LIN {X 0,Y 474.599,Z 728.17,A -85,B 0,C 180,E1 -7141.218,E2 -7141.218} C_VEL
LIN {X 0,Y 474.621,Z 728.178,A -85,B 0,C 180,E1 -7144.242,E2 -7144.242} C_VEL
LIN {X 0,Y 474.591,Z 728.17,A -85,B 0,C 180,E1 -7147.384,E2 -7147.384} C_VEL
LIN {X 0,Y 474.618,Z 728.176,A -85,B 0,C 180,E1 -7150.658,E2 -7150.658} C_VEL
LIN {X 0,Y 474.601,Z 728.174,A -85,B 0,C 180,E1 -7153.481,E2 -7153.481} C_VEL
LIN {X 0,Y 474.593,Z 728.164,A -85,B 0,C 180,E1 -7156.52,E2 -7156.52} C_VEL
LIN {X 0,Y 474.618,Z 728.164,A -85,B 0,C 180,E1 -7159.342,E2 -7159.342} C_VEL
LIN {X 0,Y 474.591,Z 728.181,A -85,B 0,C 180,E1 -7162.616,E2 -7162.616} C_VEL
LIN {X 0,Y 474.621,Z 728.167,A -85,B 0,C 180,E1 -7165.758,E2 -7165.758} C_VEL
LIN {X 0,Y 474.599,Z 728.178,A -85,B 0,C 180,E1 -7168.782,E2 -7168.782} C_VEL
LIN {X 0,Y 474.646,Z 728.168,A -85,B 0,C 180,E1 -7171.717,E2 -7171.717} C_VEL
LIN {X 0,Y 474.655,Z 728.161,A -85,B 0,C 180,E1 -7174.582,E2 -7174.582} C_VEL
LIN {X 0,Y 474.603,Z 728.179,A -85,B 0,C 180,E1 -7177.355,E2 -7177.355} C_VEL
LIN {X 0,Y 474.656,Z 728.166,A -85,B 0,C 180,E1 -7180.09,E2 -7180.09} C_VEL
LIN {X 0,Y 474.641,Z 728.164,A -85,B 0,C 180,E1 -7182.774,E2 -7182.774} C_VEL
LIN {X 0,Y 474.655,Z 728.173,A -85,B 0,C 180,E1 -7185.421,E2 -7185.421} C_VEL
LIN {X 0,Y 474.707,Z 728.161,A -85,B 0,C 180,E1 -7188.038,E2 -7188.038} C_VEL
LIN {X 0,Y 474.729,Z 728.152,A -85,B 0,C 180,E1 -7191.486,E2 -7191.486} C_VEL
LIN {X 0,Y 474.773,Z 728.149,A -85,B 0,C 180,E1 -7194.052,E2 -7194.052} C_VEL
LIN {X 0,Y 474.897,Z 728.146,A -85,B 0,C 180,E1 -7197.455,E2 -7197.455} C_VEL
LIN {X 0,Y 474.913,Z 728.132,A -85,B 0,C 180,E1 -7200,E2 -7200} C_VEL
LIN {X 0,Y 474.896,Z 728.125,A -85,B 0,C 180,E1 -7202.545,E2 -7202.545} C_VEL
LIN {X 0,Y 474.774,Z 728.157,A -85,B 0,C 180,E1 -7205.948,E2 -7205.948} C_VEL
LIN {X 0,Y 474.73,Z 728.158,A -85,B 0,C 180,E1 -7208.513,E2 -7208.513} C_VEL
LIN {X 0,Y 474.706,Z 728.156,A -85,B 0,C 180,E1 -7211.962,E2 -7211.962} C_VEL
LIN {X 0,Y 474.702,Z 728.163,A -85,B 0,C 180,E1 -7215.455,E2 -7215.455} C_VEL
LIN {X 0,Y 474.668,Z 728.164,A -85,B 0,C 180,E1 -7219.01,E2 -7219.01} C_VEL
LIN {X 0,Y 474.593,Z 728.171,A -85,B 0,C 180,E1 -7221.729,E2 -7221.729} C_VEL
LIN {X 0,Y 474.661,Z 728.169,A -85,B 0,C 180,E1 -7224.493,E2 -7224.493} C_VEL
LIN {X 0,Y 474.7,Z 728.161,A -85,B 0,C 180,E1 -7227.339,E2 -7227.339} C_VEL
LIN {X 0,Y 474.606,Z 728.172,A -85,B 0,C 180,E1 -7230.81,E2 -7230.81} C_VEL
LIN {X 0,Y 474.64,Z 728.175,A -85,B 0,C 180,E1 -7233.984,E2 -7233.984} C_VEL
LIN {X 0,Y 474.576,Z 728.167,A -85,B 0,C 180,E1 -7236.9,E2 -7236.9} C_VEL
LIN {X 0,Y 474.651,Z 728.143,A -85,B 0,C 180,E1 -7239.651,E2 -7239.651} C_VEL
LIN {X 0,Y 474.616,Z 728.173,A -85,B 0,C 180,E1 -7242.934,E2 -7242.934} C_VEL
LIN {X 0,Y 474.61,Z 728.175,A -85,B 0,C 180,E1 -7245.895,E2 -7245.895} C_VEL
LIN {X 0,Y 474.629,Z 728.168,A -85,B 0,C 180,E1 -7249.041,E2 -7249.041} C_VEL
LIN {X 0,Y 474.612,Z 728.174,A -85,B 0,C 180,E1 -7251.704,E2 -7251.704} C_VEL
LIN {X 0,Y 474.631,Z 728.174,A -85,B 0,C 180,E1 -7254.726,E2 -7254.726} C_VEL
LIN {X 0,Y 474.638,Z 728.168,A -85,B 0,C 180,E1 -7257.788,E2 -7257.788} C_VEL
LIN {X 0,Y 474.625,Z 728.176,A -85,B 0,C 180,E1 -7260.884,E2 -7260.884} C_VEL
LIN {X 0,Y 474.661,Z 728.165,A -85,B 0,C 180,E1 -7263.628,E2 -7263.628} C_VEL
LIN {X 0,Y 474.654,Z 728.288,A -85,B 0,C 180,E1 -7266.436,E2 -7266.436} C_VEL
LIN {X 0,Y 475.974,Z 735.804,A -85,B 0,C 180,E1 -7268.11,E2 -7268.11} C_VEL
LIN {X 0,Y 475.496,Z 750.231,A -85,B 0,C 180,E1 -7271.075,E2 -7271.075} C_VEL
LIN {X 0,Y 474.91,Z 765.942,A -85,B 0,C 180,E1 -7274.261,E2 -7274.261} C_VEL
LIN {X 0,Y 474.578,Z 778.638,A -85,B 0,C 180,E1 -7276.784,E2 -7276.784} C_VEL
LIN {X 0,Y 475.05,Z 782.47,A -85,B 0,C 180,E1 -7276.903,E2 -7276.903} C_VEL
LIN {X 0,Y 476.424,Z 793.246,A -85,B 0,C 180,E1 -7277.104,E2 -7277.104} C_VEL
LIN {X 0,Y 476.124,Z 856.175,A -85,B 0,C 180,E1 -7278.074,E2 -7278.074} C_VEL
LIN {X 0,Y 475.856,Z 866.65,A -85,B 0,C 180,E1 -7278.364,E2 -7278.364} C_VEL
LIN {X 0,Y 475.632,Z 877.37,A -85,B 0,C 180,E1 -7278.817,E2 -7278.817} C_VEL
LIN {X 0,Y 475.292,Z 888.005,A -85,B 0,C 180,E1 -7279.456,E2 -7279.456} C_VEL
LIN {X 0,Y 474.98,Z 896.334,A -85,B 0,C 180,E1 -7280.095,E2 -7280.095} C_VEL
LIN {X 0,Y 474.712,Z 904.218,A -85,B 0,C 180,E1 -7280.842,E2 -7280.842} C_VEL
LIN {X 0,Y 474.417,Z 911.588,A -85,B 0,C 180,E1 -7281.695,E2 -7281.695} C_VEL
LIN {X 0,Y 474.217,Z 919.07,A -85,B 0,C 180,E1 -7282.763,E2 -7282.763} C_VEL
LIN {X 0,Y 474.006,Z 925.901,A -85,B 0,C 180,E1 -7284.043,E2 -7284.043} C_VEL
LIN {X 0,Y 473.815,Z 931.085,A -85,B 0,C 180,E1 -7285.321,E2 -7285.321} C_VEL
LIN {X 0,Y 473.832,Z 934.897,A -85,B 0,C 180,E1 -7286.599,E2 -7286.599} C_VEL
LIN {X 0,Y 473.727,Z 936.647,A -85,B 0,C 180,E1 -7287.449,E2 -7287.449} C_VEL
LIN {X 0,Y 473.693,Z 937.902,A -85,B 0,C 180,E1 -7288.3,E2 -7288.3} C_VEL
LIN {X 0,Y 473.686,Z 938.684,A -85,B 0,C 180,E1 -7289.15,E2 -7289.15} C_VEL
LIN {X 0,Y 473.666,Z 938.979,A -85,B 0,C 180,E1 -7290,E2 -7290} C_VEL
LIN {X 0,Y 473.686,Z 938.683,A -85,B 0,C 180,E1 -7290.85,E2 -7290.85} C_VEL
LIN {X 0,Y 473.693,Z 937.901,A -85,B 0,C 180,E1 -7291.7,E2 -7291.7} C_VEL
LIN {X 0,Y 473.727,Z 936.646,A -85,B 0,C 180,E1 -7292.551,E2 -7292.551} C_VEL
LIN {X 0,Y 473.849,Z 933.739,A -85,B 0,C 180,E1 -7293.827,E2 -7293.827} C_VEL
LIN {X 0,Y 473.815,Z 931.085,A -85,B 0,C 180,E1 -7294.679,E2 -7294.679} C_VEL
LIN {X 0,Y 474.006,Z 925.898,A -85,B 0,C 180,E1 -7295.957,E2 -7295.957} C_VEL
LIN {X 0,Y 474.19,Z 919.063,A -85,B 0,C 180,E1 -7297.237,E2 -7297.237} C_VEL
LIN {X 0,Y 474.417,Z 911.591,A -85,B 0,C 180,E1 -7298.305,E2 -7298.305} C_VEL
LIN {X 0,Y 474.712,Z 904.224,A -85,B 0,C 180,E1 -7299.158,E2 -7299.158} C_VEL
LIN {X 0,Y 474.98,Z 896.337,A -85,B 0,C 180,E1 -7299.905,E2 -7299.905} C_VEL
LIN {X 0,Y 475.292,Z 888.006,A -85,B 0,C 180,E1 -7300.544,E2 -7300.544} C_VEL
LIN {X 0,Y 475.646,Z 877.374,A -85,B 0,C 180,E1 -7301.182,E2 -7301.182} C_VEL
LIN {X 0,Y 475.886,Z 865.822,A -85,B 0,C 180,E1 -7301.662,E2 -7301.662} C_VEL
LIN {X 0,Y 476.121,Z 856.176,A -85,B 0,C 180,E1 -7301.926,E2 -7301.926} C_VEL
LIN {X 0,Y 476.367,Z 808.389,A -85,B 0,C 180,E1 -7302.669,E2 -7302.669} C_VEL
LIN {X 0,Y 476.334,Z 792.236,A -85,B 0,C 180,E1 -7302.914,E2 -7302.914} C_VEL
LIN {X 0,Y 474.578,Z 778.937,A -85,B 0,C 180,E1 -7303.189,E2 -7303.189} C_VEL
LIN {X 0,Y 474.708,Z 773.874,A -85,B 0,C 180,E1 -7304.139,E2 -7304.139} C_VEL
LIN {X 0,Y 475.222,Z 757.609,A -85,B 0,C 180,E1 -7307.426,E2 -7307.426} C_VEL
LIN {X 0,Y 475.836,Z 741.257,A -85,B 0,C 180,E1 -7310.761,E2 -7310.761} C_VEL
LIN {X 0,Y 475.962,Z 735.791,A -85,B 0,C 180,E1 -7311.891,E2 -7311.891} C_VEL
LIN {X 0,Y 474.664,Z 728.224,A -85,B 0,C 180,E1 -7313.593,E2 -7313.593} C_VEL
LIN {X 0,Y 474.661,Z 728.165,A -85,B 0,C 180,E1 -7316.372,E2 -7316.372} C_VEL
LIN {X 0,Y 474.623,Z 728.174,A -85,B 0,C 180,E1 -7319.252,E2 -7319.252} C_VEL
LIN {X 0,Y 474.618,Z 728.171,A -85,B 0,C 180,E1 -7322.431,E2 -7322.431} C_VEL
LIN {X 0,Y 474.621,Z 728.174,A -85,B 0,C 180,E1 -7325.47,E2 -7325.47} C_VEL
LIN {X 0,Y 474.613,Z 728.173,A -85,B 0,C 180,E1 -7328.457,E2 -7328.457} C_VEL
LIN {X 0,Y 474.629,Z 728.167,A -85,B 0,C 180,E1 -7330.959,E2 -7330.959} C_VEL
LIN {X 0,Y 474.61,Z 728.175,A -85,B 0,C 180,E1 -7334.105,E2 -7334.105} C_VEL
LIN {X 0,Y 474.616,Z 728.172,A -85,B 0,C 180,E1 -7337.066,E2 -7337.066} C_VEL
LIN {X 0,Y 474.67,Z 728.139,A -85,B 0,C 180,E1 -7340.457,E2 -7340.457} C_VEL
LIN {X 0,Y 474.595,Z 728.172,A -85,B 0,C 180,E1 -7343.677,E2 -7343.677} C_VEL
LIN {X 0,Y 474.644,Z 728.169,A -85,B 0,C 180,E1 -7346.78,E2 -7346.78} C_VEL
LIN {X 0,Y 474.607,Z 728.175,A -85,B 0,C 180,E1 -7349.77,E2 -7349.77} C_VEL
LIN {X 0,Y 474.698,Z 728.162,A -85,B 0,C 180,E1 -7352.68,E2 -7352.68} C_VEL
LIN {X 0,Y 474.661,Z 728.169,A -85,B 0,C 180,E1 -7355.507,E2 -7355.507} C_VEL
LIN {X 0,Y 474.673,Z 728.156,A -85,B 0,C 180,E1 -7359.186,E2 -7359.186} C_VEL
LIN {X 0,Y 474.659,Z 728.17,A -85,B 0,C 180,E1 -7361.885,E2 -7361.885} C_VEL
LIN {X 0,Y 474.702,Z 728.163,A -85,B 0,C 180,E1 -7364.545,E2 -7364.545} C_VEL
LIN {X 0,Y 474.706,Z 728.155,A -85,B 0,C 180,E1 -7368.038,E2 -7368.038} C_VEL
LIN {X 0,Y 474.73,Z 728.157,A -85,B 0,C 180,E1 -7371.487,E2 -7371.487} C_VEL
LIN {X 0,Y 474.775,Z 728.156,A -85,B 0,C 180,E1 -7374.052,E2 -7374.052} C_VEL
LIN {X 0,Y 474.897,Z 728.124,A -85,B 0,C 180,E1 -7377.455,E2 -7377.455} C_VEL
LIN {X 0,Y 474.914,Z 728.132,A -85,B 0,C 180,E1 -7380,E2 -7380} C_VEL
LIN {X 0,Y 474.897,Z 728.145,A -85,B 0,C 180,E1 -7382.545,E2 -7382.545} C_VEL
LIN {X 0,Y 474.773,Z 728.148,A -85,B 0,C 180,E1 -7385.948,E2 -7385.948} C_VEL
LIN {X 0,Y 474.729,Z 728.151,A -85,B 0,C 180,E1 -7388.514,E2 -7388.514} C_VEL
LIN {X 0,Y 474.707,Z 728.161,A -85,B 0,C 180,E1 -7391.962,E2 -7391.962} C_VEL
LIN {X 0,Y 474.702,Z 728.157,A -85,B 0,C 180,E1 -7395.456,E2 -7395.456} C_VEL
LIN {X 0,Y 474.665,Z 728.169,A -85,B 0,C 180,E1 -7399.01,E2 -7399.01} C_VEL
LIN {X 0,Y 474.59,Z 728.176,A -85,B 0,C 180,E1 -7401.729,E2 -7401.729} C_VEL
LIN {X 0,Y 474.651,Z 728.167,A -85,B 0,C 180,E1 -7404.493,E2 -7404.493} C_VEL
LIN {X 0,Y 474.683,Z 728.167,A -85,B 0,C 180,E1 -7407.334,E2 -7407.334} C_VEL
LIN {X 0,Y 474.606,Z 728.174,A -85,B 0,C 180,E1 -7410.23,E2 -7410.23} C_VEL
LIN {X 0,Y 474.626,Z 728.171,A -85,B 0,C 180,E1 -7413.221,E2 -7413.221} C_VEL
LIN {X 0,Y 474.59,Z 728.176,A -85,B 0,C 180,E1 -7416.324,E2 -7416.324} C_VEL
LIN {X 0,Y 474.619,Z 728.168,A -85,B 0,C 180,E1 -7419.646,E2 -7419.646} C_VEL
LIN {X 0,Y 474.604,Z 728.149,A -85,B 0,C 180,E1 -7422.234,E2 -7422.234} C_VEL
LIN {X 0,Y 474.618,Z 728.17,A -85,B 0,C 180,E1 -7425.298,E2 -7425.298} C_VEL
LIN {X 0,Y 474.622,Z 728.173,A -85,B 0,C 180,E1 -7428.215,E2 -7428.215} C_VEL
LIN {X 0,Y 474.613,Z 728.168,A -85,B 0,C 180,E1 -7431.543,E2 -7431.543} C_VEL
LIN {X 0,Y 474.624,Z 728.173,A -85,B 0,C 180,E1 -7434.726,E2 -7434.726} C_VEL
LIN {X 0,Y 474.636,Z 728.169,A -85,B 0,C 180,E1 -7437.788,E2 -7437.788} C_VEL
LIN {X 0,Y 474.608,Z 728.175,A -85,B 0,C 180,E1 -7440.888,E2 -7440.888} C_VEL
LIN {X 0,Y 474.615,Z 728.18,A -85,B 0,C 180,E1 -7443.626,E2 -7443.626} C_VEL
LIN {X 0,Y 474.636,Z 728.17,A -85,B 0,C 180,E1 -7446.642,E2 -7446.642} C_VEL
LIN {X 0,Y 474.674,Z 728.172,A -85,B 0,C 180,E1 -7450.09,E2 -7450.09} C_VEL
LIN {X 0,Y 474.695,Z 728.188,A -85,B 0,C 180,E1 -7450.387,E2 -7450.387} C_VEL
LIN {X 0,Y 474.548,Z 728.717,A -85,B 0,C 180,E1 -7450.744,E2 -7450.744} C_VEL
LIN {X 0,Y 473.678,Z 730.812,A -85,B 0,C 180,E1 -7451.298,E2 -7451.298} C_VEL
LIN {X 0,Y 468.563,Z 738.885,A -85,B 0,C 180,E1 -7453.14,E2 -7453.14} C_VEL
LIN {X 0,Y 467.847,Z 741.421,A -85,B 0,C 180,E1 -7453.786,E2 -7453.786} C_VEL
LIN {X 0,Y 467.504,Z 752.277,A -85,B 0,C 180,E1 -7456.526,E2 -7456.526} C_VEL
LIN {X 0,Y 467.554,Z 753.524,A -85,B 0,C 180,E1 -7456.689,E2 -7456.689} C_VEL
LIN {X 0,Y 469.574,Z 765.597,A -85,B 0,C 180,E1 -7456.949,E2 -7456.949} C_VEL
LIN {X 0,Y 469.229,Z 828.139,A -85,B 0,C 180,E1 -7457.923,E2 -7457.923} C_VEL
LIN {X 0,Y 469.116,Z 837.235,A -85,B 0,C 180,E1 -7458.167,E2 -7458.167} C_VEL
LIN {X 0,Y 468.858,Z 846.827,A -85,B 0,C 180,E1 -7458.544,E2 -7458.544} C_VEL
LIN {X 0,Y 468.61,Z 856.862,A -85,B 0,C 180,E1 -7459.085,E2 -7459.085} C_VEL
LIN {X 0,Y 468.208,Z 867.274,A -85,B 0,C 180,E1 -7459.841,E2 -7459.841} C_VEL
LIN {X 0,Y 467.908,Z 875.411,A -85,B 0,C 180,E1 -7460.599,E2 -7460.599} C_VEL
LIN {X 0,Y 467.607,Z 882.124,A -85,B 0,C 180,E1 -7461.356,E2 -7461.356} C_VEL
LIN {X 0,Y 467.352,Z 888.477,A -85,B 0,C 180,E1 -7462.222,E2 -7462.222} C_VEL
LIN {X 0,Y 467.173,Z 894.148,A -85,B 0,C 180,E1 -7463.161,E2 -7463.161} C_VEL
LIN {X 0,Y 467.132,Z 898.161,A -85,B 0,C 180,E1 -7463.955,E2 -7463.955} C_VEL
LIN {X 0,Y 466.829,Z 901.837,A -85,B 0,C 180,E1 -7464.817,E2 -7464.817} C_VEL
LIN {X 0,Y 466.84,Z 904.829,A -85,B 0,C 180,E1 -7465.683,E2 -7465.683} C_VEL
LIN {X 0,Y 466.793,Z 907.149,A -85,B 0,C 180,E1 -7466.547,E2 -7466.547} C_VEL
LIN {X 0,Y 466.687,Z 908.919,A -85,B 0,C 180,E1 -7467.411,E2 -7467.411} C_VEL
LIN {X 0,Y 466.634,Z 910.196,A -85,B 0,C 180,E1 -7468.274,E2 -7468.274} C_VEL
LIN {X 0,Y 466.617,Z 911.003,A -85,B 0,C 180,E1 -7469.137,E2 -7469.137} C_VEL
LIN {X 0,Y 466.597,Z 911.311,A -85,B 0,C 180,E1 -7470,E2 -7470} C_VEL
LIN {X 0,Y 466.617,Z 911.037,A -85,B 0,C 180,E1 -7470.863,E2 -7470.863} C_VEL
LIN {X 0,Y 466.634,Z 910.296,A -85,B 0,C 180,E1 -7471.726,E2 -7471.726} C_VEL
LIN {X 0,Y 466.687,Z 909.088,A -85,B 0,C 180,E1 -7472.589,E2 -7472.589} C_VEL
LIN {X 0,Y 466.841,Z 906.243,A -85,B 0,C 180,E1 -7473.884,E2 -7473.884} C_VEL
LIN {X 0,Y 466.806,Z 903.66,A -85,B 0,C 180,E1 -7474.75,E2 -7474.75} C_VEL
LIN {X 0,Y 467.107,Z 898.559,A -85,B 0,C 180,E1 -7476.046,E2 -7476.046} C_VEL
LIN {X 0,Y 467.194,Z 893.079,A -85,B 0,C 180,E1 -7477.129,E2 -7477.129} C_VEL
LIN {X 0,Y 467.46,Z 886.192,A -85,B 0,C 180,E1 -7478.211,E2 -7478.211} C_VEL
LIN {X 0,Y 467.806,Z 878.281,A -85,B 0,C 180,E1 -7479.185,E2 -7479.185} C_VEL
LIN {X 0,Y 468.108,Z 870.734,A -85,B 0,C 180,E1 -7479.942,E2 -7479.942} C_VEL
LIN {X 0,Y 468.366,Z 862.827,A -85,B 0,C 180,E1 -7480.592,E2 -7480.592} C_VEL
LIN {X 0,Y 468.66,Z 854.66,A -85,B 0,C 180,E1 -7481.132,E2 -7481.132} C_VEL
LIN {X 0,Y 468.943,Z 846.391,A -85,B 0,C 180,E1 -7481.563,E2 -7481.563} C_VEL
LIN {X 0,Y 469.105,Z 837.469,A -85,B 0,C 180,E1 -7481.915,E2 -7481.915} C_VEL
LIN {X 0,Y 469.271,Z 828.375,A -85,B 0,C 180,E1 -7482.161,E2 -7482.161} C_VEL
LIN {X 0,Y 469.463,Z 764.852,A -85,B 0,C 180,E1 -7483.156,E2 -7483.156} C_VEL
LIN {X 0,Y 467.486,Z 752.928,A -85,B 0,C 180,E1 -7483.398,E2 -7483.398} C_VEL
LIN {X 0,Y 467.842,Z 741.837,A -85,B 0,C 180,E1 -7486.197,E2 -7486.197} C_VEL
LIN {X 0,Y 468.105,Z 733.408,A -85,B 0,C 180,E1 -7488.378,E2 -7488.378} C_VEL
LIN {X 0,Y 467.664,Z 729.117,A -85,B 0,C 180,E1 -7489.591,E2 -7489.591} C_VEL
LIN {X 0,Y 467.577,Z 729.049,A -85,B 0,C 180,E1 -7493.004,E2 -7493.004} C_VEL
LIN {X 0,Y 467.569,Z 729.056,A -85,B 0,C 180,E1 -7495.842,E2 -7495.842} C_VEL
LIN {X 0,Y 467.555,Z 729.056,A -85,B 0,C 180,E1 -7498.751,E2 -7498.751} C_VEL
LIN {X 0,Y 467.583,Z 729.045,A -85,B 0,C 180,E1 -7501.74,E2 -7501.74} C_VEL
LIN {X 0,Y 467.56,Z 729.057,A -85,B 0,C 180,E1 -7504.833,E2 -7504.833} C_VEL
LIN {X 0,Y 467.565,Z 729.047,A -85,B 0,C 180,E1 -7508.045,E2 -7508.045} C_VEL
LIN {X 0,Y 467.579,Z 729.05,A -85,B 0,C 180,E1 -7511.277,E2 -7511.277} C_VEL
LIN {X 0,Y 467.553,Z 729.052,A -85,B 0,C 180,E1 -7513.821,E2 -7513.821} C_VEL
LIN {X 0,Y 467.55,Z 729.046,A -85,B 0,C 180,E1 -7516.255,E2 -7516.255} C_VEL
LIN {X 0,Y 467.576,Z 729.04,A -85,B 0,C 180,E1 -7519.735,E2 -7519.735} C_VEL
LIN {X 0,Y 467.549,Z 729.061,A -85,B 0,C 180,E1 -7522.814,E2 -7522.814} C_VEL
LIN {X 0,Y 467.578,Z 729.045,A -85,B 0,C 180,E1 -7525.76,E2 -7525.76} C_VEL
LIN {X 0,Y 467.569,Z 729.057,A -85,B 0,C 180,E1 -7528.955,E2 -7528.955} C_VEL
LIN {X 0,Y 467.635,Z 729.042,A -85,B 0,C 180,E1 -7532.462,E2 -7532.462} C_VEL
LIN {X 0,Y 467.596,Z 729.046,A -85,B 0,C 180,E1 -7535.112,E2 -7535.112} C_VEL
LIN {X 0,Y 467.536,Z 729.055,A -85,B 0,C 180,E1 -7537.926,E2 -7537.926} C_VEL
LIN {X 0,Y 467.624,Z 729.044,A -85,B 0,C 180,E1 -7540.692,E2 -7540.692} C_VEL
LIN {X 0,Y 467.651,Z 729.034,A -85,B 0,C 180,E1 -7544.115,E2 -7544.115} C_VEL
LIN {X 0,Y 467.656,Z 729.043,A -85,B 0,C 180,E1 -7547.642,E2 -7547.642} C_VEL
LIN {X 0,Y 467.663,Z 729.034,A -85,B 0,C 180,E1 -7550.485,E2 -7550.485} C_VEL
LIN {X 0,Y 467.702,Z 729.024,A -85,B 0,C 180,E1 -7553.095,E2 -7553.095} C_VEL
LIN {X 0,Y 467.726,Z 729.027,A -85,B 0,C 180,E1 -7554.827,E2 -7554.827} C_VEL
LIN {X 0,Y 467.862,Z 729.021,A -85,B 0,C 180,E1 -7557.417,E2 -7557.417} C_VEL
LIN {X 0,Y 467.884,Z 729.008,A -85,B 0,C 180,E1 -7560,E2 -7560} C_VEL
LIN {X 0,Y 467.861,Z 729,A -85,B 0,C 180,E1 -7562.583,E2 -7562.583} C_VEL
LIN {X 0,Y 467.739,Z 729.032,A -85,B 0,C 180,E1 -7566.037,E2 -7566.037} C_VEL
LIN {X 0,Y 467.684,Z 729.035,A -85,B 0,C 180,E1 -7568.643,E2 -7568.643} C_VEL
LIN {X 0,Y 467.658,Z 729.032,A -85,B 0,C 180,E1 -7572.145,E2 -7572.145} C_VEL
LIN {X 0,Y 467.641,Z 729.045,A -85,B 0,C 180,E1 -7575.695,E2 -7575.695} C_VEL
LIN {X 0,Y 467.62,Z 729.042,A -85,B 0,C 180,E1 -7578.765,E2 -7578.765} C_VEL
LIN {X 0,Y 467.583,Z 729.04,A -85,B 0,C 180,E1 -7581.268,E2 -7581.268} C_VEL
LIN {X 0,Y 467.576,Z 729.053,A -85,B 0,C 180,E1 -7583.943,E2 -7583.943} C_VEL
LIN {X 0,Y 467.618,Z 729.044,A -85,B 0,C 180,E1 -7586.8,E2 -7586.8} C_VEL
LIN {X 0,Y 467.555,Z 729.047,A -85,B 0,C 180,E1 -7589.738,E2 -7589.738} C_VEL
LIN {X 0,Y 467.585,Z 729.05,A -85,B 0,C 180,E1 -7592.758,E2 -7592.758} C_VEL
LIN {X 0,Y 467.558,Z 729.053,A -85,B 0,C 180,E1 -7595.889,E2 -7595.889} C_VEL
LIN {X 0,Y 467.601,Z 729.019,A -85,B 0,C 180,E1 -7599.143,E2 -7599.143} C_VEL
LIN {X 0,Y 467.587,Z 729.05,A -85,B 0,C 180,E1 -7602.567,E2 -7602.567} C_VEL
LIN {X 0,Y 467.571,Z 729.051,A -85,B 0,C 180,E1 -7605.053,E2 -7605.053} C_VEL
LIN {X 0,Y 467.589,Z 729.042,A -85,B 0,C 180,E1 -7607.44,E2 -7607.44} C_VEL
LIN {X 0,Y 467.593,Z 729.052,A -85,B 0,C 180,E1 -7610.856,E2 -7610.856} C_VEL
LIN {X 0,Y 467.564,Z 729.051,A -85,B 0,C 180,E1 -7614.26,E2 -7614.26} C_VEL
LIN {X 0,Y 467.583,Z 729.047,A -85,B 0,C 180,E1 -7617.321,E2 -7617.321} C_VEL
LIN {X 0,Y 467.571,Z 729.05,A -85,B 0,C 180,E1 -7620.667,E2 -7620.667} C_VEL
LIN {X 0,Y 467.616,Z 729.042,A -85,B 0,C 180,E1 -7623.2,E2 -7623.2} C_VEL
LIN {X 0,Y 467.633,Z 729.209,A -85,B 0,C 180,E1 -7626.305,E2 -7626.305} C_VEL
LIN {X 0,Y 468.955,Z 736.728,A -85,B 0,C 180,E1 -7627.996,E2 -7627.996} C_VEL
LIN {X 0,Y 468.526,Z 749.812,A -85,B 0,C 180,E1 -7630.731,E2 -7630.731} C_VEL
LIN {X 0,Y 467.915,Z 765.671,A -85,B 0,C 180,E1 -7634.001,E2 -7634.001} C_VEL
LIN {X 0,Y 467.541,Z 778.521,A -85,B 0,C 180,E1 -7636.591,E2 -7636.591} C_VEL
LIN {X 0,Y 468.158,Z 783.277,A -85,B 0,C 180,E1 -7636.722,E2 -7636.722} C_VEL
LIN {X 0,Y 469.509,Z 795.019,A -85,B 0,C 180,E1 -7636.941,E2 -7636.941} C_VEL
LIN {X 0,Y 469.185,Z 855.966,A -85,B 0,C 180,E1 -7637.895,E2 -7637.895} C_VEL
LIN {X 0,Y 468.922,Z 866.441,A -85,B 0,C 180,E1 -7638.19,E2 -7638.19} C_VEL
LIN {X 0,Y 468.651,Z 877.161,A -85,B 0,C 180,E1 -7638.649,E2 -7638.649} C_VEL
LIN {X 0,Y 468.295,Z 887.796,A -85,B 0,C 180,E1 -7639.297,E2 -7639.297} C_VEL
LIN {X 0,Y 467.965,Z 896.124,A -85,B 0,C 180,E1 -7639.945,E2 -7639.945} C_VEL
LIN {X 0,Y 467.673,Z 904.008,A -85,B 0,C 180,E1 -7640.703,E2 -7640.703} C_VEL
LIN {X 0,Y 467.368,Z 911.379,A -85,B 0,C 180,E1 -7641.569,E2 -7641.569} C_VEL
LIN {X 0,Y 467.143,Z 918.86,A -85,B 0,C 180,E1 -7642.653,E2 -7642.653} C_VEL
LIN {X 0,Y 466.916,Z 925.691,A -85,B 0,C 180,E1 -7643.952,E2 -7643.952} C_VEL
LIN {X 0,Y 466.739,Z 930.876,A -85,B 0,C 180,E1 -7645.249,E2 -7645.249} C_VEL
LIN {X 0,Y 466.734,Z 934.687,A -85,B 0,C 180,E1 -7646.547,E2 -7646.547} C_VEL
LIN {X 0,Y 466.65,Z 936.438,A -85,B 0,C 180,E1 -7647.41,E2 -7647.41} C_VEL
LIN {X 0,Y 466.603,Z 937.693,A -85,B 0,C 180,E1 -7648.274,E2 -7648.274} C_VEL
LIN {X 0,Y 466.616,Z 938.476,A -85,B 0,C 180,E1 -7649.137,E2 -7649.137} C_VEL
LIN {X 0,Y 466.596,Z 938.771,A -85,B 0,C 180,E1 -7650,E2 -7650} C_VEL
LIN {X 0,Y 466.616,Z 938.475,A -85,B 0,C 180,E1 -7650.863,E2 -7650.863} C_VEL
LIN {X 0,Y 466.603,Z 937.692,A -85,B 0,C 180,E1 -7651.726,E2 -7651.726} C_VEL
LIN {X 0,Y 466.65,Z 936.437,A -85,B 0,C 180,E1 -7652.59,E2 -7652.59} C_VEL
LIN {X 0,Y 466.74,Z 933.529,A -85,B 0,C 180,E1 -7653.885,E2 -7653.885} C_VEL
LIN {X 0,Y 466.739,Z 930.876,A -85,B 0,C 180,E1 -7654.751,E2 -7654.751} C_VEL
LIN {X 0,Y 466.917,Z 925.688,A -85,B 0,C 180,E1 -7656.048,E2 -7656.048} C_VEL
LIN {X 0,Y 467.132,Z 918.853,A -85,B 0,C 180,E1 -7657.347,E2 -7657.347} C_VEL
LIN {X 0,Y 467.368,Z 911.381,A -85,B 0,C 180,E1 -7658.431,E2 -7658.431} C_VEL
LIN {X 0,Y 467.673,Z 904.015,A -85,B 0,C 180,E1 -7659.297,E2 -7659.297} C_VEL
LIN {X 0,Y 467.965,Z 896.127,A -85,B 0,C 180,E1 -7660.055,E2 -7660.055} C_VEL
LIN {X 0,Y 468.297,Z 887.797,A -85,B 0,C 180,E1 -7660.703,E2 -7660.703} C_VEL
LIN {X 0,Y 468.697,Z 877.166,A -85,B 0,C 180,E1 -7661.35,E2 -7661.35} C_VEL
LIN {X 0,Y 468.932,Z 865.613,A -85,B 0,C 180,E1 -7661.838,E2 -7661.838} C_VEL
LIN {X 0,Y 469.195,Z 855.968,A -85,B 0,C 180,E1 -7662.105,E2 -7662.105} C_VEL
LIN {X 0,Y 469.455,Z 793.148,A -85,B 0,C 180,E1 -7663.089,E2 -7663.089} C_VEL
LIN {X 0,Y 467.567,Z 778.882,A -85,B 0,C 180,E1 -7663.381,E2 -7663.381} C_VEL
LIN {X 0,Y 467.58,Z 776.934,A -85,B 0,C 180,E1 -7663.694,E2 -7663.694} C_VEL
LIN {X 0,Y 468.085,Z 761.783,A -85,B 0,C 180,E1 -7666.8,E2 -7666.8} C_VEL
LIN {X 0,Y 468.663,Z 746.541,A -85,B 0,C 180,E1 -7669.947,E2 -7669.947} C_VEL
LIN {X 0,Y 468.933,Z 736.714,A -85,B 0,C 180,E1 -7672.005,E2 -7672.005} C_VEL
LIN {X 0,Y 467.633,Z 729.106,A -85,B 0,C 180,E1 -7673.741,E2 -7673.741} C_VEL
LIN {X 0,Y 467.616,Z 729.042,A -85,B 0,C 180,E1 -7676.8,E2 -7676.8} C_VEL
LIN {X 0,Y 467.555,Z 729.047,A -85,B 0,C 180,E1 -7679.738,E2 -7679.738} C_VEL
LIN {X 0,Y 467.584,Z 729.049,A -85,B 0,C 180,E1 -7682.758,E2 -7682.758} C_VEL
LIN {X 0,Y 467.558,Z 729.051,A -85,B 0,C 180,E1 -7685.889,E2 -7685.889} C_VEL
LIN {X 0,Y 467.593,Z 729.052,A -85,B 0,C 180,E1 -7689.144,E2 -7689.144} C_VEL
LIN {X 0,Y 467.587,Z 729.043,A -85,B 0,C 180,E1 -7692.567,E2 -7692.567} C_VEL
LIN {X 0,Y 467.571,Z 729.052,A -85,B 0,C 180,E1 -7695.053,E2 -7695.053} C_VEL
LIN {X 0,Y 467.589,Z 729.05,A -85,B 0,C 180,E1 -7697.44,E2 -7697.44} C_VEL
LIN {X 0,Y 467.601,Z 729.018,A -85,B 0,C 180,E1 -7700.857,E2 -7700.857} C_VEL
LIN {X 0,Y 467.564,Z 729.051,A -85,B 0,C 180,E1 -7704.26,E2 -7704.26} C_VEL
LIN {X 0,Y 467.583,Z 729.051,A -85,B 0,C 180,E1 -7707.321,E2 -7707.321} C_VEL
LIN {X 0,Y 467.571,Z 729.043,A -85,B 0,C 180,E1 -7710.668,E2 -7710.668} C_VEL
LIN {X 0,Y 467.618,Z 729.044,A -85,B 0,C 180,E1 -7713.2,E2 -7713.2} C_VEL
LIN {X 0,Y 467.595,Z 729.045,A -85,B 0,C 180,E1 -7716.468,E2 -7716.468} C_VEL
LIN {X 0,Y 467.626,Z 729.038,A -85,B 0,C 180,E1 -7719.777,E2 -7719.777} C_VEL
LIN {X 0,Y 467.612,Z 729.049,A -85,B 0,C 180,E1 -7722.507,E2 -7722.507} C_VEL
LIN {X 0,Y 467.608,Z 729.042,A -85,B 0,C 180,E1 -7725.197,E2 -7725.197} C_VEL
LIN {X 0,Y 467.658,Z 729.031,A -85,B 0,C 180,E1 -7727.855,E2 -7727.855} C_VEL
LIN {X 0,Y 467.684,Z 729.035,A -85,B 0,C 180,E1 -7731.357,E2 -7731.357} C_VEL
LIN {X 0,Y 467.739,Z 729.032,A -85,B 0,C 180,E1 -7733.963,E2 -7733.963} C_VEL
LIN {X 0,Y 467.862,Z 729,A -85,B 0,C 180,E1 -7737.417,E2 -7737.417} C_VEL
LIN {X 0,Y 467.885,Z 729.007,A -85,B 0,C 180,E1 -7740,E2 -7740} C_VEL
LIN {X 0,Y 467.863,Z 729.022,A -85,B 0,C 180,E1 -7742.583,E2 -7742.583} C_VEL
LIN {X 0,Y 467.737,Z 729.025,A -85,B 0,C 180,E1 -7746.038,E2 -7746.038} C_VEL
LIN {X 0,Y 467.682,Z 729.031,A -85,B 0,C 180,E1 -7748.643,E2 -7748.643} C_VEL
LIN {X 0,Y 467.658,Z 729.04,A -85,B 0,C 180,E1 -7752.145,E2 -7752.145} C_VEL
LIN {X 0,Y 467.641,Z 729.035,A -85,B 0,C 180,E1 -7755.695,E2 -7755.695} C_VEL
LIN {X 0,Y 467.615,Z 729.042,A -85,B 0,C 180,E1 -7758.763,E2 -7758.763} C_VEL
LIN {X 0,Y 467.582,Z 729.053,A -85,B 0,C 180,E1 -7761.268,E2 -7761.268} C_VEL
LIN {X 0,Y 467.569,Z 729.047,A -85,B 0,C 180,E1 -7763.944,E2 -7763.944} C_VEL
LIN {X 0,Y 467.615,Z 729.04,A -85,B 0,C 180,E1 -7766.8,E2 -7766.8} C_VEL
LIN {X 0,Y 467.555,Z 729.053,A -85,B 0,C 180,E1 -7769.738,E2 -7769.738} C_VEL
LIN {X 0,Y 467.58,Z 729.048,A -85,B 0,C 180,E1 -7772.759,E2 -7772.759} C_VEL
LIN {X 0,Y 467.554,Z 729.053,A -85,B 0,C 180,E1 -7775.89,E2 -7775.89} C_VEL
LIN {X 0,Y 467.577,Z 729.053,A -85,B 0,C 180,E1 -7779.145,E2 -7779.145} C_VEL
LIN {X 0,Y 467.577,Z 729.033,A -85,B 0,C 180,E1 -7781.403,E2 -7781.403} C_VEL
LIN {X 0,Y 467.567,Z 729.045,A -85,B 0,C 180,E1 -7785.053,E2 -7785.053} C_VEL
LIN {X 0,Y 467.59,Z 729.055,A -85,B 0,C 180,E1 -7787.44,E2 -7787.44} C_VEL
LIN {X 0,Y 467.561,Z 729.045,A -85,B 0,C 180,E1 -7790.853,E2 -7790.853} C_VEL
LIN {X 0,Y 467.56,Z 729.055,A -85,B 0,C 180,E1 -7794.261,E2 -7794.261} C_VEL
LIN {X 0,Y 467.581,Z 729.053,A -85,B 0,C 180,E1 -7797.321,E2 -7797.321} C_VEL
LIN {X 0,Y 467.558,Z 729.053,A -85,B 0,C 180,E1 -7800.67,E2 -7800.67} C_VEL
LIN {X 0,Y 467.565,Z 729.053,A -85,B 0,C 180,E1 -7803.196,E2 -7803.196} C_VEL
LIN {X 0,Y 467.591,Z 729.048,A -85,B 0,C 180,E1 -7806.469,E2 -7806.469} C_VEL
LIN {X 0,Y 467.635,Z 729.05,A -85,B 0,C 180,E1 -7809.778,E2 -7809.778} C_VEL
LIN {X 0,Y 467.716,Z 729.213,A -85,B 0,C 180,E1 -7810.582,E2 -7810.582} C_VEL
LIN {X 0,Y 468.082,Z 734.779,A -85,B 0,C 180,E1 -7812.073,E2 -7812.073} C_VEL
LIN {X 0,Y 467.847,Z 741.421,A -85,B 0,C 180,E1 -7813.786,E2 -7813.786} C_VEL
LIN {X 0,Y 467.125,Z 743.198,A -85,B 0,C 180,E1 -7814.214,E2 -7814.214} C_VEL
LIN {X 0,Y 464.196,Z 746.192,A -85,B 0,C 180,E1 -7814.864,E2 -7814.864} C_VEL
LIN {X 0,Y 461.251,Z 749.201,A -85,B 0,C 180,E1 -7815.52,E2 -7815.52} C_VEL
LIN {X 0,Y 460.519,Z 751.004,A -85,B 0,C 180,E1 -7815.953,E2 -7815.953} C_VEL
LIN {X 0,Y 460.516,Z 753.153,A -85,B 0,C 180,E1 -7816.441,E2 -7816.441} C_VEL
LIN {X 0,Y 461.216,Z 757.471,A -85,B 0,C 180,E1 -7816.576,E2 -7816.576} C_VEL
LIN {X 0,Y 462.71,Z 766.919,A -85,B 0,C 180,E1 -7816.769,E2 -7816.769} C_VEL
LIN {X 0,Y 462.301,Z 828.374,A -85,B 0,C 180,E1 -7817.74,E2 -7817.74} C_VEL
LIN {X 0,Y 462.198,Z 837.461,A -85,B 0,C 180,E1 -7817.987,E2 -7817.987} C_VEL
LIN {X 0,Y 461.905,Z 847.048,A -85,B 0,C 180,E1 -7818.369,E2 -7818.369} C_VEL
LIN {X 0,Y 461.648,Z 857.08,A -85,B 0,C 180,E1 -7818.919,E2 -7818.919} C_VEL
LIN {X 0,Y 461.235,Z 867.489,A -85,B 0,C 180,E1 -7819.686,E2 -7819.686} C_VEL
LIN {X 0,Y 460.922,Z 875.625,A -85,B 0,C 180,E1 -7820.455,E2 -7820.455} C_VEL
LIN {X 0,Y 460.582,Z 882.338,A -85,B 0,C 180,E1 -7821.223,E2 -7821.223} C_VEL
LIN {X 0,Y 460.335,Z 888.69,A -85,B 0,C 180,E1 -7822.102,E2 -7822.102} C_VEL
LIN {X 0,Y 460.112,Z 894.822,A -85,B 0,C 180,E1 -7823.142,E2 -7823.142} C_VEL
LIN {X 0,Y 460.073,Z 898.372,A -85,B 0,C 180,E1 -7823.862,E2 -7823.862} C_VEL
LIN {X 0,Y 459.777,Z 902.048,A -85,B 0,C 180,E1 -7824.738,E2 -7824.738} C_VEL
LIN {X 0,Y 459.748,Z 905.041,A -85,B 0,C 180,E1 -7825.616,E2 -7825.616} C_VEL
LIN {X 0,Y 459.732,Z 907.359,A -85,B 0,C 180,E1 -7826.494,E2 -7826.494} C_VEL
LIN {X 0,Y 459.611,Z 909.129,A -85,B 0,C 180,E1 -7827.371,E2 -7827.371} C_VEL
LIN {X 0,Y 459.545,Z 910.405,A -85,B 0,C 180,E1 -7828.247,E2 -7828.247} C_VEL
LIN {X 0,Y 459.521,Z 911.212,A -85,B 0,C 180,E1 -7829.124,E2 -7829.124} C_VEL
LIN {X 0,Y 459.528,Z 911.519,A -85,B 0,C 180,E1 -7830,E2 -7830} C_VEL
LIN {X 0,Y 459.521,Z 911.245,A -85,B 0,C 180,E1 -7830.876,E2 -7830.876} C_VEL
LIN {X 0,Y 459.546,Z 910.504,A -85,B 0,C 180,E1 -7831.753,E2 -7831.753} C_VEL
LIN {X 0,Y 459.611,Z 909.295,A -85,B 0,C 180,E1 -7832.629,E2 -7832.629} C_VEL
LIN {X 0,Y 459.774,Z 906.45,A -85,B 0,C 180,E1 -7833.944,E2 -7833.944} C_VEL
LIN {X 0,Y 459.724,Z 903.867,A -85,B 0,C 180,E1 -7834.823,E2 -7834.823} C_VEL
LIN {X 0,Y 460.062,Z 898.765,A -85,B 0,C 180,E1 -7836.139,E2 -7836.139} C_VEL
LIN {X 0,Y 460.149,Z 893.284,A -85,B 0,C 180,E1 -7837.239,E2 -7837.239} C_VEL
LIN {X 0,Y 460.441,Z 886.397,A -85,B 0,C 180,E1 -7838.338,E2 -7838.338} C_VEL
LIN {X 0,Y 460.81,Z 878.483,A -85,B 0,C 180,E1 -7839.326,E2 -7839.326} C_VEL
LIN {X 0,Y 461.104,Z 870.937,A -85,B 0,C 180,E1 -7840.095,E2 -7840.095} C_VEL
LIN {X 0,Y 461.39,Z 863.028,A -85,B 0,C 180,E1 -7840.754,E2 -7840.754} C_VEL
LIN {X 0,Y 461.703,Z 854.859,A -85,B 0,C 180,E1 -7841.302,E2 -7841.302} C_VEL
LIN {X 0,Y 461.993,Z 846.587,A -85,B 0,C 180,E1 -7841.74,E2 -7841.74} C_VEL
LIN {X 0,Y 462.181,Z 837.66,A -85,B 0,C 180,E1 -7842.097,E2 -7842.097} C_VEL
LIN {X 0,Y 462.346,Z 828.659,A -85,B 0,C 180,E1 -7842.343,E2 -7842.343} C_VEL
LIN {X 0,Y 462.613,Z 765.973,A -85,B 0,C 180,E1 -7843.339,E2 -7843.339} C_VEL
LIN {X 0,Y 460.479,Z 752.975,A -85,B 0,C 180,E1 -7843.632,E2 -7843.632} C_VEL
LIN {X 0,Y 460.856,Z 742.21,A -85,B 0,C 180,E1 -7846.393,E2 -7846.393} C_VEL
LIN {X 0,Y 461.049,Z 733.57,A -85,B 0,C 180,E1 -7848.67,E2 -7848.67} C_VEL
LIN {X 0,Y 460.627,Z 730.016,A -85,B 0,C 180,E1 -7849.671,E2 -7849.671} C_VEL
LIN {X 0,Y 460.545,Z 729.925,A -85,B 0,C 180,E1 -7853.376,E2 -7853.376} C_VEL
LIN {X 0,Y 460.521,Z 729.935,A -85,B 0,C 180,E1 -7856.268,E2 -7856.268} C_VEL
LIN {X 0,Y 460.527,Z 729.929,A -85,B 0,C 180,E1 -7859.232,E2 -7859.232} C_VEL
LIN {X 0,Y 460.531,Z 729.925,A -85,B 0,C 180,E1 -7862.284,E2 -7862.284} C_VEL
LIN {X 0,Y 460.509,Z 729.932,A -85,B 0,C 180,E1 -7865.446,E2 -7865.446} C_VEL
LIN {X 0,Y 460.534,Z 729.921,A -85,B 0,C 180,E1 -7868.896,E2 -7868.896} C_VEL
LIN {X 0,Y 460.524,Z 729.931,A -85,B 0,C 180,E1 -7872.181,E2 -7872.181} C_VEL
LIN {X 0,Y 460.514,Z 729.921,A -85,B 0,C 180,E1 -7875.411,E2 -7875.411} C_VEL
LIN {X 0,Y 460.531,Z 729.917,A -85,B 0,C 180,E1 -7878.989,E2 -7878.989} C_VEL
LIN {X 0,Y 460.525,Z 729.929,A -85,B 0,C 180,E1 -7881.267,E2 -7881.267} C_VEL
LIN {X 0,Y 460.509,Z 729.935,A -85,B 0,C 180,E1 -7884.554,E2 -7884.554} C_VEL
LIN {X 0,Y 460.531,Z 729.923,A -85,B 0,C 180,E1 -7887.715,E2 -7887.715} C_VEL
LIN {X 0,Y 460.54,Z 729.932,A -85,B 0,C 180,E1 -7890.769,E2 -7890.769} C_VEL
LIN {X 0,Y 460.56,Z 729.914,A -85,B 0,C 180,E1 -7893.734,E2 -7893.734} C_VEL
LIN {X 0,Y 460.548,Z 729.924,A -85,B 0,C 180,E1 -7896.624,E2 -7896.624} C_VEL
LIN {X 0,Y 460.553,Z 729.926,A -85,B 0,C 180,E1 -7899.453,E2 -7899.453} C_VEL
LIN {X 0,Y 460.552,Z 729.915,A -85,B 0,C 180,E1 -7902.23,E2 -7902.23} C_VEL
LIN {X 0,Y 460.57,Z 729.92,A -85,B 0,C 180,E1 -7904.965,E2 -7904.965} C_VEL
LIN {X 0,Y 460.612,Z 729.917,A -85,B 0,C 180,E1 -7908.559,E2 -7908.559} C_VEL
LIN {X 0,Y 460.697,Z 729.892,A -85,B 0,C 180,E1 -7912.108,E2 -7912.108} C_VEL
LIN {X 0,Y 460.698,Z 729.902,A -85,B 0,C 180,E1 -7914.748,E2 -7914.748} C_VEL
LIN {X 0,Y 460.827,Z 729.897,A -85,B 0,C 180,E1 -7917.378,E2 -7917.378} C_VEL
LIN {X 0,Y 460.854,Z 729.883,A -85,B 0,C 180,E1 -7920,E2 -7920} C_VEL
LIN {X 0,Y 460.802,Z 729.879,A -85,B 0,C 180,E1 -7922.622,E2 -7922.622} C_VEL
LIN {X 0,Y 460.705,Z 729.908,A -85,B 0,C 180,E1 -7926.13,E2 -7926.13} C_VEL
LIN {X 0,Y 460.631,Z 729.914,A -85,B 0,C 180,E1 -7928.776,E2 -7928.776} C_VEL
LIN {X 0,Y 460.615,Z 729.906,A -85,B 0,C 180,E1 -7932.445,E2 -7932.445} C_VEL
LIN {X 0,Y 460.602,Z 729.925,A -85,B 0,C 180,E1 -7935.997,E2 -7935.997} C_VEL
LIN {X 0,Y 460.573,Z 729.919,A -85,B 0,C 180,E1 -7938.902,E2 -7938.902} C_VEL
LIN {X 0,Y 460.518,Z 729.921,A -85,B 0,C 180,E1 -7941.485,E2 -7941.485} C_VEL
LIN {X 0,Y 460.545,Z 729.93,A -85,B 0,C 180,E1 -7944.332,E2 -7944.332} C_VEL
LIN {X 0,Y 460.58,Z 729.92,A -85,B 0,C 180,E1 -7947.243,E2 -7947.243} C_VEL
LIN {X 0,Y 460.512,Z 729.93,A -85,B 0,C 180,E1 -7950.24,E2 -7950.24} C_VEL
LIN {X 0,Y 460.531,Z 729.928,A -85,B 0,C 180,E1 -7953.325,E2 -7953.325} C_VEL
LIN {X 0,Y 460.48,Z 729.925,A -85,B 0,C 180,E1 -7956.529,E2 -7956.529} C_VEL
LIN {X 0,Y 460.575,Z 729.895,A -85,B 0,C 180,E1 -7959.858,E2 -7959.858} C_VEL
LIN {X 0,Y 460.514,Z 729.93,A -85,B 0,C 180,E1 -7962.9,E2 -7962.9} C_VEL
LIN {X 0,Y 460.512,Z 729.931,A -85,B 0,C 180,E1 -7965.83,E2 -7965.83} C_VEL
LIN {X 0,Y 460.533,Z 729.923,A -85,B 0,C 180,E1 -7968.989,E2 -7968.989} C_VEL
LIN {X 0,Y 460.532,Z 729.929,A -85,B 0,C 180,E1 -7971.267,E2 -7971.267} C_VEL
LIN {X 0,Y 460.514,Z 729.93,A -85,B 0,C 180,E1 -7974.555,E2 -7974.555} C_VEL
LIN {X 0,Y 460.533,Z 729.925,A -85,B 0,C 180,E1 -7977.716,E2 -7977.716} C_VEL
LIN {X 0,Y 460.541,Z 729.927,A -85,B 0,C 180,E1 -7980.769,E2 -7980.769} C_VEL
LIN {X 0,Y 460.563,Z 729.92,A -85,B 0,C 180,E1 -7983.735,E2 -7983.735} C_VEL
LIN {X 0,Y 460.584,Z 730.001,A -85,B 0,C 180,E1 -7986.109,E2 -7986.109} C_VEL
LIN {X 0,Y 462.013,Z 738.714,A -85,B 0,C 180,E1 -7988.112,E2 -7988.112} C_VEL
LIN {X 0,Y 461.431,Z 752.63,A -85,B 0,C 180,E1 -7991.057,E2 -7991.057} C_VEL
LIN {X 0,Y 460.847,Z 767.001,A -85,B 0,C 180,E1 -7994.068,E2 -7994.068} C_VEL
LIN {X 0,Y 460.54,Z 778.382,A -85,B 0,C 180,E1 -7996.388,E2 -7996.388} C_VEL
LIN {X 0,Y 461.34,Z 784.613,A -85,B 0,C 180,E1 -7996.546,E2 -7996.546} C_VEL
LIN {X 0,Y 462.604,Z 794.93,A -85,B 0,C 180,E1 -7996.744,E2 -7996.744} C_VEL
LIN {X 0,Y 462.254,Z 855.762,A -85,B 0,C 180,E1 -7997.71,E2 -7997.71} C_VEL
LIN {X 0,Y 461.992,Z 866.236,A -85,B 0,C 180,E1 -7998.01,E2 -7998.01} C_VEL
LIN {X 0,Y 461.697,Z 876.953,A -85,B 0,C 180,E1 -7998.475,E2 -7998.475} C_VEL
LIN {X 0,Y 461.317,Z 887.587,A -85,B 0,C 180,E1 -7999.133,E2 -7999.133} C_VEL
LIN {X 0,Y 460.965,Z 895.916,A -85,B 0,C 180,E1 -7999.791,E2 -7999.791} C_VEL
LIN {X 0,Y 460.627,Z 903.798,A -85,B 0,C 180,E1 -8000.56,E2 -8000.56} C_VEL
LIN {X 0,Y 460.333,Z 911.169,A -85,B 0,C 180,E1 -8001.439,E2 -8001.439} C_VEL
LIN {X 0,Y 460.074,Z 918.65,A -85,B 0,C 180,E1 -8002.539,E2 -8002.539} C_VEL
LIN {X 0,Y 459.83,Z 925.481,A -85,B 0,C 180,E1 -8003.858,E2 -8003.858} C_VEL
LIN {X 0,Y 459.668,Z 930.668,A -85,B 0,C 180,E1 -8005.176,E2 -8005.176} C_VEL
LIN {X 0,Y 459.634,Z 934.478,A -85,B 0,C 180,E1 -8006.494,E2 -8006.494} C_VEL
LIN {X 0,Y 459.575,Z 936.23,A -85,B 0,C 180,E1 -8007.371,E2 -8007.371} C_VEL
LIN {X 0,Y 459.515,Z 937.484,A -85,B 0,C 180,E1 -8008.247,E2 -8008.247} C_VEL
LIN {X 0,Y 459.519,Z 938.267,A -85,B 0,C 180,E1 -8009.124,E2 -8009.124} C_VEL
LIN {X 0,Y 459.527,Z 938.563,A -85,B 0,C 180,E1 -8010,E2 -8010} C_VEL
LIN {X 0,Y 459.519,Z 938.266,A -85,B 0,C 180,E1 -8010.876,E2 -8010.876} C_VEL
LIN {X 0,Y 459.515,Z 937.484,A -85,B 0,C 180,E1 -8011.753,E2 -8011.753} C_VEL
LIN {X 0,Y 459.575,Z 936.229,A -85,B 0,C 180,E1 -8012.629,E2 -8012.629} C_VEL
LIN {X 0,Y 459.633,Z 933.32,A -85,B 0,C 180,E1 -8013.945,E2 -8013.945} C_VEL
LIN {X 0,Y 459.668,Z 930.667,A -85,B 0,C 180,E1 -8014.824,E2 -8014.824} C_VEL
LIN {X 0,Y 459.831,Z 925.479,A -85,B 0,C 180,E1 -8016.142,E2 -8016.142} C_VEL
LIN {X 0,Y 460.07,Z 918.644,A -85,B 0,C 180,E1 -8017.461,E2 -8017.461} C_VEL
LIN {X 0,Y 460.333,Z 911.171,A -85,B 0,C 180,E1 -8018.561,E2 -8018.561} C_VEL
LIN {X 0,Y 460.627,Z 903.804,A -85,B 0,C 180,E1 -8019.44,E2 -8019.44} C_VEL
LIN {X 0,Y 460.965,Z 895.918,A -85,B 0,C 180,E1 -8020.209,E2 -8020.209} C_VEL
LIN {X 0,Y 461.32,Z 887.587,A -85,B 0,C 180,E1 -8020.867,E2 -8020.867} C_VEL
LIN {X 0,Y 461.752,Z 876.956,A -85,B 0,C 180,E1 -8021.523,E2 -8021.523} C_VEL
LIN {X 0,Y 461.973,Z 865.401,A -85,B 0,C 180,E1 -8022.019,E2 -8022.019} C_VEL
LIN {X 0,Y 462.268,Z 855.755,A -85,B 0,C 180,E1 -8022.289,E2 -8022.289} C_VEL
LIN {X 0,Y 462.534,Z 793.804,A -85,B 0,C 180,E1 -8023.275,E2 -8023.275} C_VEL
LIN {X 0,Y 460.53,Z 778.678,A -85,B 0,C 180,E1 -8023.589,E2 -8023.589} C_VEL
LIN {X 0,Y 460.548,Z 776.736,A -85,B 0,C 180,E1 -8023.907,E2 -8023.907} C_VEL
LIN {X 0,Y 461.108,Z 761.599,A -85,B 0,C 180,E1 -8027.062,E2 -8027.062} C_VEL
LIN {X 0,Y 461.742,Z 745.273,A -85,B 0,C 180,E1 -8030.492,E2 -8030.492} C_VEL
LIN {X 0,Y 461.948,Z 737.912,A -85,B 0,C 180,E1 -8032.061,E2 -8032.061} C_VEL
LIN {X 0,Y 460.584,Z 729.997,A -85,B 0,C 180,E1 -8033.891,E2 -8033.891} C_VEL
LIN {X 0,Y 460.58,Z 729.921,A -85,B 0,C 180,E1 -8037.243,E2 -8037.243} C_VEL
LIN {X 0,Y 460.512,Z 729.921,A -85,B 0,C 180,E1 -8040.24,E2 -8040.24} C_VEL
LIN {X 0,Y 460.53,Z 729.934,A -85,B 0,C 180,E1 -8043.325,E2 -8043.325} C_VEL
LIN {X 0,Y 460.48,Z 729.93,A -85,B 0,C 180,E1 -8046.529,E2 -8046.529} C_VEL
LIN {X 0,Y 460.567,Z 729.92,A -85,B 0,C 180,E1 -8049.859,E2 -8049.859} C_VEL
LIN {X 0,Y 460.513,Z 729.925,A -85,B 0,C 180,E1 -8052.9,E2 -8052.9} C_VEL
LIN {X 0,Y 460.512,Z 729.933,A -85,B 0,C 180,E1 -8055.83,E2 -8055.83} C_VEL
LIN {X 0,Y 460.54,Z 729.915,A -85,B 0,C 180,E1 -8058.99,E2 -8058.99} C_VEL
LIN {X 0,Y 460.54,Z 729.899,A -85,B 0,C 180,E1 -8061.268,E2 -8061.268} C_VEL
LIN {X 0,Y 460.515,Z 729.927,A -85,B 0,C 180,E1 -8064.555,E2 -8064.555} C_VEL
LIN {X 0,Y 460.533,Z 729.934,A -85,B 0,C 180,E1 -8067.716,E2 -8067.716} C_VEL
LIN {X 0,Y 460.541,Z 729.918,A -85,B 0,C 180,E1 -8070.769,E2 -8070.769} C_VEL
LIN {X 0,Y 460.564,Z 729.927,A -85,B 0,C 180,E1 -8073.735,E2 -8073.735} C_VEL
LIN {X 0,Y 460.548,Z 729.922,A -85,B 0,C 180,E1 -8076.624,E2 -8076.624} C_VEL
LIN {X 0,Y 460.554,Z 729.915,A -85,B 0,C 180,E1 -8079.453,E2 -8079.453} C_VEL
LIN {X 0,Y 460.562,Z 729.931,A -85,B 0,C 180,E1 -8082.23,E2 -8082.23} C_VEL
LIN {X 0,Y 460.567,Z 729.92,A -85,B 0,C 180,E1 -8084.965,E2 -8084.965} C_VEL
LIN {X 0,Y 460.613,Z 729.914,A -85,B 0,C 180,E1 -8088.559,E2 -8088.559} C_VEL
LIN {X 0,Y 460.697,Z 729.911,A -85,B 0,C 180,E1 -8092.109,E2 -8092.109} C_VEL
LIN {X 0,Y 460.698,Z 729.905,A -85,B 0,C 180,E1 -8094.748,E2 -8094.748} C_VEL
LIN {X 0,Y 460.803,Z 729.879,A -85,B 0,C 180,E1 -8097.378,E2 -8097.378} C_VEL
LIN {X 0,Y 460.856,Z 729.883,A -85,B 0,C 180,E1 -8100,E2 -8100} C_VEL
LIN {X 0,Y 460.827,Z 729.897,A -85,B 0,C 180,E1 -8102.622,E2 -8102.622} C_VEL
LIN {X 0,Y 460.704,Z 729.902,A -85,B 0,C 180,E1 -8106.13,E2 -8106.13} C_VEL
LIN {X 0,Y 460.629,Z 729.911,A -85,B 0,C 180,E1 -8108.776,E2 -8108.776} C_VEL
LIN {X 0,Y 460.615,Z 729.92,A -85,B 0,C 180,E1 -8112.445,E2 -8112.445} C_VEL
LIN {X 0,Y 460.602,Z 729.912,A -85,B 0,C 180,E1 -8115.998,E2 -8115.998} C_VEL
LIN {X 0,Y 460.57,Z 729.921,A -85,B 0,C 180,E1 -8119.616,E2 -8119.616} C_VEL
LIN {X 0,Y 460.512,Z 729.931,A -85,B 0,C 180,E1 -8122.429,E2 -8122.429} C_VEL
LIN {X 0,Y 460.556,Z 729.914,A -85,B 0,C 180,E1 -8125.799,E2 -8125.799} C_VEL
LIN {X 0,Y 460.554,Z 729.922,A -85,B 0,C 180,E1 -8128.233,E2 -8128.233} C_VEL
LIN {X 0,Y 460.521,Z 729.931,A -85,B 0,C 180,E1 -8131.283,E2 -8131.283} C_VEL
LIN {X 0,Y 460.524,Z 729.924,A -85,B 0,C 180,E1 -8134.504,E2 -8134.504} C_VEL
LIN {X 0,Y 460.502,Z 729.933,A -85,B 0,C 180,E1 -8137.623,E2 -8137.623} C_VEL
LIN {X 0,Y 460.54,Z 729.917,A -85,B 0,C 180,E1 -8140.269,E2 -8140.269} C_VEL
LIN {X 0,Y 460.51,Z 729.911,A -85,B 0,C 180,E1 -8143.374,E2 -8143.374} C_VEL
LIN {X 0,Y 460.497,Z 729.931,A -85,B 0,C 180,E1 -8146.624,E2 -8146.624} C_VEL
LIN {X 0,Y 460.54,Z 729.924,A -85,B 0,C 180,E1 -8149.731,E2 -8149.731} C_VEL
LIN {X 0,Y 460.501,Z 729.924,A -85,B 0,C 180,E1 -8152.524,E2 -8152.524} C_VEL
LIN {X 0,Y 460.538,Z 729.936,A -85,B 0,C 180,E1 -8155.623,E2 -8155.623} C_VEL
LIN {X 0,Y 460.539,Z 729.92,A -85,B 0,C 180,E1 -8158.745,E2 -8158.745} C_VEL
LIN {X 0,Y 460.552,Z 729.928,A -85,B 0,C 180,E1 -8162.261,E2 -8162.261} C_VEL
LIN {X 0,Y 460.535,Z 729.928,A -85,B 0,C 180,E1 -8164.704,E2 -8164.704} C_VEL
LIN {X 0,Y 460.512,Z 729.933,A -85,B 0,C 180,E1 -8167.571,E2 -8167.571} C_VEL
LIN {X 0,Y 460.661,Z 730.119,A -85,B 0,C 180,E1 -8170.476,E2 -8170.476} C_VEL
LIN {X 0,Y 461.099,Z 734.944,A -85,B 0,C 180,E1 -8171.793,E2 -8171.793} C_VEL
LIN {X 0,Y 460.661,Z 747.147,A -85,B 0,C 180,E1 -8174.968,E2 -8174.968} C_VEL
LIN {X 0,Y 460.519,Z 751.004,A -85,B 0,C 180,E1 -8175.953,E2 -8175.953} C_VEL
LIN {X 0,Y 460.057,Z 752.709,A -85,B 0,C 180,E1 -8176.203,E2 -8176.203} C_VEL
LIN {X 0,Y 458.688,Z 755.778,A -85,B 0,C 180,E1 -8176.394,E2 -8176.394} C_VEL
LIN {X 0,Y 456.6,Z 760.284,A -85,B 0,C 180,E1 -8176.479,E2 -8176.479} C_VEL
LIN {X 0,Y 455.362,Z 764.157,A -85,B 0,C 180,E1 -8176.503,E2 -8176.503} C_VEL
LIN {X 0,Y 454.924,Z 768.499,A -85,B 0,C 180,E1 -8176.554,E2 -8176.554} C_VEL
LIN {X 0,Y 455.664,Z 781.624,A -85,B 0,C 180,E1 -8176.79,E2 -8176.79} C_VEL
LIN {X 0,Y 455.386,Z 828.606,A -85,B 0,C 180,E1 -8177.55,E2 -8177.55} C_VEL
LIN {X 0,Y 455.28,Z 837.684,A -85,B 0,C 180,E1 -8177.802,E2 -8177.802} C_VEL
LIN {X 0,Y 454.961,Z 847.268,A -85,B 0,C 180,E1 -8178.189,E2 -8178.189} C_VEL
LIN {X 0,Y 454.691,Z 857.298,A -85,B 0,C 180,E1 -8178.747,E2 -8178.747} C_VEL
LIN {X 0,Y 454.276,Z 867.703,A -85,B 0,C 180,E1 -8179.526,E2 -8179.526} C_VEL
LIN {X 0,Y 453.939,Z 875.839,A -85,B 0,C 180,E1 -8180.307,E2 -8180.307} C_VEL
LIN {X 0,Y 453.578,Z 882.551,A -85,B 0,C 180,E1 -8181.086,E2 -8181.086} C_VEL
LIN {X 0,Y 453.301,Z 888.902,A -85,B 0,C 180,E1 -8181.979,E2 -8181.979} C_VEL
LIN {X 0,Y 453.096,Z 894.18,A -85,B 0,C 180,E1 -8182.872,E2 -8182.872} C_VEL
LIN {X 0,Y 453.023,Z 898.583,A -85,B 0,C 180,E1 -8183.766,E2 -8183.766} C_VEL
LIN {X 0,Y 452.655,Z 903.768,A -85,B 0,C 180,E1 -8185.101,E2 -8185.101} C_VEL
LIN {X 0,Y 452.709,Z 906.424,A -85,B 0,C 180,E1 -8185.994,E2 -8185.994} C_VEL
LIN {X 0,Y 452.539,Z 909.338,A -85,B 0,C 180,E1 -8187.33,E2 -8187.33} C_VEL
LIN {X 0,Y 452.46,Z 910.615,A -85,B 0,C 180,E1 -8188.22,E2 -8188.22} C_VEL
LIN {X 0,Y 452.428,Z 911.421,A -85,B 0,C 180,E1 -8189.11,E2 -8189.11} C_VEL
LIN {X 0,Y 452.433,Z 911.728,A -85,B 0,C 180,E1 -8190,E2 -8190} C_VEL
LIN {X 0,Y 452.428,Z 911.454,A -85,B 0,C 180,E1 -8190.89,E2 -8190.89} C_VEL
LIN {X 0,Y 452.461,Z 910.712,A -85,B 0,C 180,E1 -8191.78,E2 -8191.78} C_VEL
LIN {X 0,Y 452.539,Z 909.503,A -85,B 0,C 180,E1 -8192.67,E2 -8192.67} C_VEL
LIN {X 0,Y 452.706,Z 906.657,A -85,B 0,C 180,E1 -8194.006,E2 -8194.006} C_VEL
LIN {X 0,Y 452.65,Z 904.074,A -85,B 0,C 180,E1 -8194.899,E2 -8194.899} C_VEL
LIN {X 0,Y 452.999,Z 898.972,A -85,B 0,C 180,E1 -8196.235,E2 -8196.235} C_VEL
LIN {X 0,Y 453.094,Z 893.491,A -85,B 0,C 180,E1 -8197.352,E2 -8197.352} C_VEL
LIN {X 0,Y 453.413,Z 886.602,A -85,B 0,C 180,E1 -8198.468,E2 -8198.468} C_VEL
LIN {X 0,Y 453.796,Z 878.688,A -85,B 0,C 180,E1 -8199.471,E2 -8199.471} C_VEL
LIN {X 0,Y 454.118,Z 871.14,A -85,B 0,C 180,E1 -8200.252,E2 -8200.252} C_VEL
LIN {X 0,Y 454.422,Z 863.229,A -85,B 0,C 180,E1 -8200.921,E2 -8200.921} C_VEL
LIN {X 0,Y 454.751,Z 855.059,A -85,B 0,C 180,E1 -8201.477,E2 -8201.477} C_VEL
LIN {X 0,Y 455.059,Z 846.784,A -85,B 0,C 180,E1 -8201.921,E2 -8201.921} C_VEL
LIN {X 0,Y 455.268,Z 837.853,A -85,B 0,C 180,E1 -8202.283,E2 -8202.283} C_VEL
LIN {X 0,Y 455.446,Z 828.107,A -85,B 0,C 180,E1 -8202.549,E2 -8202.549} C_VEL
LIN {X 0,Y 455.662,Z 766.27,A -85,B 0,C 180,E1 -8203.545,E2 -8203.545} C_VEL
LIN {X 0,Y 453.457,Z 753.174,A -85,B 0,C 180,E1 -8203.846,E2 -8203.846} C_VEL
LIN {X 0,Y 453.95,Z 740.656,A -85,B 0,C 180,E1 -8207.107,E2 -8207.107} C_VEL
LIN {X 0,Y 453.921,Z 732.953,A -85,B 0,C 180,E1 -8209.186,E2 -8209.186} C_VEL
LIN {X 0,Y 453.582,Z 730.877,A -85,B 0,C 180,E1 -8209.823,E2 -8209.823} C_VEL
LIN {X 0,Y 453.48,Z 730.807,A -85,B 0,C 180,E1 -8212.796,E2 -8212.796} C_VEL
LIN {X 0,Y 453.486,Z 730.81,A -85,B 0,C 180,E1 -8215.99,E2 -8215.99} C_VEL
LIN {X 0,Y 453.493,Z 730.808,A -85,B 0,C 180,E1 -8218.713,E2 -8218.713} C_VEL
LIN {X 0,Y 453.464,Z 730.803,A -85,B 0,C 180,E1 -8221.8,E2 -8221.8} C_VEL
LIN {X 0,Y 453.478,Z 730.81,A -85,B 0,C 180,E1 -8224.99,E2 -8224.99} C_VEL
LIN {X 0,Y 453.461,Z 730.8,A -85,B 0,C 180,E1 -8228.312,E2 -8228.312} C_VEL
LIN {X 0,Y 453.495,Z 730.805,A -85,B 0,C 180,E1 -8230.609,E2 -8230.609} C_VEL
LIN {X 0,Y 453.456,Z 730.809,A -85,B 0,C 180,E1 -8233.244,E2 -8233.244} C_VEL
LIN {X 0,Y 453.462,Z 730.798,A -85,B 0,C 180,E1 -8235.778,E2 -8235.778} C_VEL
LIN {X 0,Y 453.495,Z 730.794,A -85,B 0,C 180,E1 -8239.409,E2 -8239.409} C_VEL
LIN {X 0,Y 453.45,Z 730.809,A -85,B 0,C 180,E1 -8242.227,E2 -8242.227} C_VEL
LIN {X 0,Y 453.483,Z 730.803,A -85,B 0,C 180,E1 -8245.224,E2 -8245.224} C_VEL
LIN {X 0,Y 453.466,Z 730.806,A -85,B 0,C 180,E1 -8248.475,E2 -8248.475} C_VEL
LIN {X 0,Y 453.533,Z 730.797,A -85,B 0,C 180,E1 -8252.041,E2 -8252.041} C_VEL
LIN {X 0,Y 453.509,Z 730.802,A -85,B 0,C 180,E1 -8255.265,E2 -8255.265} C_VEL
LIN {X 0,Y 453.482,Z 730.806,A -85,B 0,C 180,E1 -8258.415,E2 -8258.415} C_VEL
LIN {X 0,Y 453.524,Z 730.802,A -85,B 0,C 180,E1 -8261.009,E2 -8261.009} C_VEL
LIN {X 0,Y 453.571,Z 730.788,A -85,B 0,C 180,E1 -8263.88,E2 -8263.88} C_VEL
LIN {X 0,Y 453.565,Z 730.8,A -85,B 0,C 180,E1 -8267.471,E2 -8267.471} C_VEL
LIN {X 0,Y 453.593,Z 730.791,A -85,B 0,C 180,E1 -8271.087,E2 -8271.087} C_VEL
LIN {X 0,Y 453.671,Z 730.779,A -85,B 0,C 180,E1 -8273.775,E2 -8273.775} C_VEL
LIN {X 0,Y 453.768,Z 730.775,A -85,B 0,C 180,E1 -8277.337,E2 -8277.337} C_VEL
LIN {X 0,Y 453.825,Z 730.758,A -85,B 0,C 180,E1 -8280,E2 -8280} C_VEL
LIN {X 0,Y 453.746,Z 730.758,A -85,B 0,C 180,E1 -8282.663,E2 -8282.663} C_VEL
LIN {X 0,Y 453.673,Z 730.783,A -85,B 0,C 180,E1 -8286.225,E2 -8286.225} C_VEL
LIN {X 0,Y 453.594,Z 730.791,A -85,B 0,C 180,E1 -8288.913,E2 -8288.913} C_VEL
LIN {X 0,Y 453.565,Z 730.784,A -85,B 0,C 180,E1 -8292.529,E2 -8292.529} C_VEL
LIN {X 0,Y 453.546,Z 730.801,A -85,B 0,C 180,E1 -8296.196,E2 -8296.196} C_VEL
LIN {X 0,Y 453.523,Z 730.798,A -85,B 0,C 180,E1 -8299.041,E2 -8299.041} C_VEL
LIN {X 0,Y 453.479,Z 730.8,A -85,B 0,C 180,E1 -8301.836,E2 -8301.836} C_VEL
LIN {X 0,Y 453.516,Z 730.802,A -85,B 0,C 180,E1 -8304.734,E2 -8304.734} C_VEL
LIN {X 0,Y 453.539,Z 730.8,A -85,B 0,C 180,E1 -8307.961,E2 -8307.961} C_VEL
LIN {X 0,Y 453.467,Z 730.806,A -85,B 0,C 180,E1 -8311.525,E2 -8311.525} C_VEL
LIN {X 0,Y 453.491,Z 730.803,A -85,B 0,C 180,E1 -8314.778,E2 -8314.778} C_VEL
LIN {X 0,Y 453.482,Z 730.783,A -85,B 0,C 180,E1 -8318.31,E2 -8318.31} C_VEL
LIN {X 0,Y 453.516,Z 730.785,A -85,B 0,C 180,E1 -8320.606,E2 -8320.606} C_VEL
LIN {X 0,Y 453.467,Z 730.811,A -85,B 0,C 180,E1 -8324.221,E2 -8324.221} C_VEL
LIN {X 0,Y 453.463,Z 730.803,A -85,B 0,C 180,E1 -8327.005,E2 -8327.005} C_VEL
LIN {X 0,Y 453.523,Z 730.804,A -85,B 0,C 180,E1 -8330.554,E2 -8330.554} C_VEL
LIN {X 0,Y 453.458,Z 730.805,A -85,B 0,C 180,E1 -8333.917,E2 -8333.917} C_VEL
LIN {X 0,Y 453.484,Z 730.805,A -85,B 0,C 180,E1 -8337.151,E2 -8337.151} C_VEL
LIN {X 0,Y 453.476,Z 730.8,A -85,B 0,C 180,E1 -8340.268,E2 -8340.268} C_VEL
LIN {X 0,Y 453.509,Z 730.798,A -85,B 0,C 180,E1 -8343.294,E2 -8343.294} C_VEL
LIN {X 0,Y 453.553,Z 730.901,A -85,B 0,C 180,E1 -8345.961,E2 -8345.961} C_VEL
LIN {X 0,Y 455.012,Z 739.348,A -85,B 0,C 180,E1 -8347.933,E2 -8347.933} C_VEL
LIN {X 0,Y 454.465,Z 752.369,A -85,B 0,C 180,E1 -8350.738,E2 -8350.738} C_VEL
LIN {X 0,Y 453.851,Z 766.812,A -85,B 0,C 180,E1 -8353.815,E2 -8353.815} C_VEL
LIN {X 0,Y 453.486,Z 778.183,A -85,B 0,C 180,E1 -8356.172,E2 -8356.172} C_VEL
LIN {X 0,Y 454.255,Z 784.203,A -85,B 0,C 180,E1 -8356.329,E2 -8356.329} C_VEL
LIN {X 0,Y 455.689,Z 796.529,A -85,B 0,C 180,E1 -8356.568,E2 -8356.568} C_VEL
LIN {X 0,Y 455.32,Z 855.561,A -85,B 0,C 180,E1 -8357.52,E2 -8357.52} C_VEL
LIN {X 0,Y 455.056,Z 866.032,A -85,B 0,C 180,E1 -8357.824,E2 -8357.824} C_VEL
LIN {X 0,Y 454.744,Z 876.748,A -85,B 0,C 180,E1 -8358.297,E2 -8358.297} C_VEL
LIN {X 0,Y 454.345,Z 887.381,A -85,B 0,C 180,E1 -8358.964,E2 -8358.964} C_VEL
LIN {X 0,Y 453.988,Z 895.709,A -85,B 0,C 180,E1 -8359.632,E2 -8359.632} C_VEL
LIN {X 0,Y 453.608,Z 903.59,A -85,B 0,C 180,E1 -8360.412,E2 -8360.412} C_VEL
LIN {X 0,Y 453.288,Z 910.961,A -85,B 0,C 180,E1 -8361.305,E2 -8361.305} C_VEL
LIN {X 0,Y 453.004,Z 918.441,A -85,B 0,C 180,E1 -8362.422,E2 -8362.422} C_VEL
LIN {X 0,Y 452.745,Z 925.272,A -85,B 0,C 180,E1 -8363.762,E2 -8363.762} C_VEL
LIN {X 0,Y 452.598,Z 930.459,A -85,B 0,C 180,E1 -8365.101,E2 -8365.101} C_VEL
LIN {X 0,Y 452.534,Z 934.269,A -85,B 0,C 180,E1 -8366.438,E2 -8366.438} C_VEL
LIN {X 0,Y 452.502,Z 936.022,A -85,B 0,C 180,E1 -8367.329,E2 -8367.329} C_VEL
LIN {X 0,Y 452.432,Z 937.276,A -85,B 0,C 180,E1 -8368.22,E2 -8368.22} C_VEL
LIN {X 0,Y 452.426,Z 938.058,A -85,B 0,C 180,E1 -8369.11,E2 -8369.11} C_VEL
LIN {X 0,Y 452.431,Z 938.354,A -85,B 0,C 180,E1 -8370,E2 -8370} C_VEL
LIN {X 0,Y 452.426,Z 938.058,A -85,B 0,C 180,E1 -8370.89,E2 -8370.89} C_VEL
LIN {X 0,Y 452.432,Z 937.275,A -85,B 0,C 180,E1 -8371.78,E2 -8371.78} C_VEL
LIN {X 0,Y 452.502,Z 936.02,A -85,B 0,C 180,E1 -8372.671,E2 -8372.671} C_VEL
LIN {X 0,Y 452.531,Z 933.11,A -85,B 0,C 180,E1 -8374.007,E2 -8374.007} C_VEL
LIN {X 0,Y 452.598,Z 930.458,A -85,B 0,C 180,E1 -8374.899,E2 -8374.899} C_VEL
LIN {X 0,Y 452.745,Z 925.268,A -85,B 0,C 180,E1 -8376.238,E2 -8376.238} C_VEL
LIN {X 0,Y 453.001,Z 918.433,A -85,B 0,C 180,E1 -8377.578,E2 -8377.578} C_VEL
LIN {X 0,Y 453.288,Z 910.961,A -85,B 0,C 180,E1 -8378.695,E2 -8378.695} C_VEL
LIN {X 0,Y 453.608,Z 903.593,A -85,B 0,C 180,E1 -8379.588,E2 -8379.588} C_VEL
LIN {X 0,Y 453.988,Z 895.707,A -85,B 0,C 180,E1 -8380.368,E2 -8380.368} C_VEL
LIN {X 0,Y 454.342,Z 887.376,A -85,B 0,C 180,E1 -8381.036,E2 -8381.036} C_VEL
LIN {X 0,Y 454.81,Z 876.744,A -85,B 0,C 180,E1 -8381.702,E2 -8381.702} C_VEL
LIN {X 0,Y 455.042,Z 865.187,A -85,B 0,C 180,E1 -8382.204,E2 -8382.204} C_VEL
LIN {X 0,Y 455.342,Z 855.538,A -85,B 0,C 180,E1 -8382.479,E2 -8382.479} C_VEL
LIN {X 0,Y 455.712,Z 796.434,A -85,B 0,C 180,E1 -8383.432,E2 -8383.432} C_VEL
LIN {X 0,Y 453.517,Z 778.475,A -85,B 0,C 180,E1 -8383.804,E2 -8383.804} C_VEL
LIN {X 0,Y 453.523,Z 776.536,A -85,B 0,C 180,E1 -8384.127,E2 -8384.127} C_VEL
LIN {X 0,Y 454.114,Z 761.414,A -85,B 0,C 180,E1 -8387.333,E2 -8387.333} C_VEL
LIN {X 0,Y 454.759,Z 746.189,A -85,B 0,C 180,E1 -8390.584,E2 -8390.584} C_VEL
LIN {X 0,Y 454.998,Z 739.355,A -85,B 0,C 180,E1 -8392.063,E2 -8392.063} C_VEL
LIN {X 0,Y 453.539,Z 730.845,A -85,B 0,C 180,E1 -8394.068,E2 -8394.068} C_VEL
LIN {X 0,Y 453.509,Z 730.798,A -85,B 0,C 180,E1 -8396.706,E2 -8396.706} C_VEL
LIN {X 0,Y 453.476,Z 730.8,A -85,B 0,C 180,E1 -8399.732,E2 -8399.732} C_VEL
LIN {X 0,Y 453.491,Z 730.809,A -85,B 0,C 180,E1 -8403.189,E2 -8403.189} C_VEL
LIN {X 0,Y 453.457,Z 730.805,A -85,B 0,C 180,E1 -8406.3,E2 -8406.3} C_VEL
LIN {X 0,Y 453.523,Z 730.803,A -85,B 0,C 180,E1 -8409.446,E2 -8409.446} C_VEL
LIN {X 0,Y 453.463,Z 730.803,A -85,B 0,C 180,E1 -8412.995,E2 -8412.995} C_VEL
LIN {X 0,Y 453.467,Z 730.811,A -85,B 0,C 180,E1 -8415.779,E2 -8415.779} C_VEL
LIN {X 0,Y 453.517,Z 730.784,A -85,B 0,C 180,E1 -8419.406,E2 -8419.406} C_VEL
LIN {X 0,Y 453.477,Z 730.796,A -85,B 0,C 180,E1 -8422.223,E2 -8422.223} C_VEL
LIN {X 0,Y 453.491,Z 730.803,A -85,B 0,C 180,E1 -8425.222,E2 -8425.222} C_VEL
LIN {X 0,Y 453.467,Z 730.805,A -85,B 0,C 180,E1 -8428.475,E2 -8428.475} C_VEL
LIN {X 0,Y 453.539,Z 730.801,A -85,B 0,C 180,E1 -8432.039,E2 -8432.039} C_VEL
LIN {X 0,Y 453.516,Z 730.801,A -85,B 0,C 180,E1 -8435.266,E2 -8435.266} C_VEL
LIN {X 0,Y 453.482,Z 730.798,A -85,B 0,C 180,E1 -8438.415,E2 -8438.415} C_VEL
LIN {X 0,Y 453.524,Z 730.798,A -85,B 0,C 180,E1 -8441.009,E2 -8441.009} C_VEL
LIN {X 0,Y 453.57,Z 730.798,A -85,B 0,C 180,E1 -8443.88,E2 -8443.88} C_VEL
LIN {X 0,Y 453.565,Z 730.783,A -85,B 0,C 180,E1 -8447.471,E2 -8447.471} C_VEL
LIN {X 0,Y 453.594,Z 730.791,A -85,B 0,C 180,E1 -8451.087,E2 -8451.087} C_VEL
LIN {X 0,Y 453.673,Z 730.782,A -85,B 0,C 180,E1 -8453.775,E2 -8453.775} C_VEL
LIN {X 0,Y 453.747,Z 730.757,A -85,B 0,C 180,E1 -8457.337,E2 -8457.337} C_VEL
LIN {X 0,Y 453.826,Z 730.758,A -85,B 0,C 180,E1 -8460,E2 -8460} C_VEL
LIN {X 0,Y 453.768,Z 730.776,A -85,B 0,C 180,E1 -8462.663,E2 -8462.663} C_VEL
LIN {X 0,Y 453.672,Z 730.779,A -85,B 0,C 180,E1 -8466.225,E2 -8466.225} C_VEL
LIN {X 0,Y 453.593,Z 730.789,A -85,B 0,C 180,E1 -8468.913,E2 -8468.913} C_VEL
LIN {X 0,Y 453.565,Z 730.8,A -85,B 0,C 180,E1 -8472.529,E2 -8472.529} C_VEL
LIN {X 0,Y 453.546,Z 730.791,A -85,B 0,C 180,E1 -8476.196,E2 -8476.196} C_VEL
LIN {X 0,Y 453.519,Z 730.802,A -85,B 0,C 180,E1 -8479.04,E2 -8479.04} C_VEL
LIN {X 0,Y 453.478,Z 730.806,A -85,B 0,C 180,E1 -8481.836,E2 -8481.836} C_VEL
LIN {X 0,Y 453.506,Z 730.803,A -85,B 0,C 180,E1 -8484.735,E2 -8484.735} C_VEL
LIN {X 0,Y 453.534,Z 730.797,A -85,B 0,C 180,E1 -8487.96,E2 -8487.96} C_VEL
LIN {X 0,Y 453.466,Z 730.807,A -85,B 0,C 180,E1 -8491.525,E2 -8491.525} C_VEL
LIN {X 0,Y 453.483,Z 730.802,A -85,B 0,C 180,E1 -8494.776,E2 -8494.776} C_VEL
LIN {X 0,Y 453.464,Z 730.806,A -85,B 0,C 180,E1 -8498.312,E2 -8498.312} C_VEL
LIN {X 0,Y 453.495,Z 730.794,A -85,B 0,C 180,E1 -8500.609,E2 -8500.609} C_VEL
LIN {X 0,Y 453.462,Z 730.798,A -85,B 0,C 180,E1 -8504.222,E2 -8504.222} C_VEL
LIN {X 0,Y 453.462,Z 730.81,A -85,B 0,C 180,E1 -8507.005,E2 -8507.005} C_VEL
LIN {X 0,Y 453.495,Z 730.807,A -85,B 0,C 180,E1 -8509.409,E2 -8509.409} C_VEL
LIN {X 0,Y 453.45,Z 730.803,A -85,B 0,C 180,E1 -8512.227,E2 -8512.227} C_VEL
LIN {X 0,Y 453.483,Z 730.81,A -85,B 0,C 180,E1 -8515.224,E2 -8515.224} C_VEL
LIN {X 0,Y 453.466,Z 730.802,A -85,B 0,C 180,E1 -8518.475,E2 -8518.475} C_VEL
LIN {X 0,Y 453.493,Z 730.807,A -85,B 0,C 180,E1 -8521.287,E2 -8521.287} C_VEL
LIN {X 0,Y 453.506,Z 730.807,A -85,B 0,C 180,E1 -8524.284,E2 -8524.284} C_VEL
LIN {X 0,Y 453.48,Z 730.806,A -85,B 0,C 180,E1 -8527.204,E2 -8527.204} C_VEL
LIN {X 0,Y 453.603,Z 730.968,A -85,B 0,C 180,E1 -8530.342,E2 -8530.342} C_VEL
LIN {X 0,Y 454.066,Z 735.111,A -85,B 0,C 180,E1 -8531.5,E2 -8531.5} C_VEL
LIN {X 0,Y 453.771,Z 745.571,A -85,B 0,C 180,E1 -8534.274,E2 -8534.274} C_VEL
LIN {X 0,Y 453.486,Z 753.351,A -85,B 0,C 180,E1 -8536.227,E2 -8536.227} C_VEL
LIN {X 0,Y 454.283,Z 758.089,A -85,B 0,C 180,E1 -8536.373,E2 -8536.373} C_VEL
LIN {X 0,Y 455.788,Z 767.884,A -85,B 0,C 180,E1 -8536.576,E2 -8536.576} C_VEL
LIN {X 0,Y 455.664,Z 781.624,A -85,B 0,C 180,E1 -8536.79,E2 -8536.79} C_VEL
LIN {X 0,Y 454.959,Z 787.465,A -85,B 0,C 180,E1 -8536.862,E2 -8536.862} C_VEL
LIN {X 0,Y 449.324,Z 806.45,A -85,B 0,C 180,E1 -8536.996,E2 -8536.996} C_VEL
LIN {X 0,Y 448.638,Z 812.291,A -85,B 0,C 180,E1 -8537.07,E2 -8537.07} C_VEL
LIN {X 0,Y 448.48,Z 830.132,A -85,B 0,C 180,E1 -8537.384,E2 -8537.384} C_VEL
LIN {X 0,Y 448.295,Z 841.222,A -85,B 0,C 180,E1 -8537.724,E2 -8537.724} C_VEL
LIN {X 0,Y 447.892,Z 851.91,A -85,B 0,C 180,E1 -8538.23,E2 -8538.23} C_VEL
LIN {X 0,Y 447.566,Z 862.241,A -85,B 0,C 180,E1 -8538.91,E2 -8538.91} C_VEL
LIN {X 0,Y 447.231,Z 870.37,A -85,B 0,C 180,E1 -8539.588,E2 -8539.588} C_VEL
LIN {X 0,Y 446.829,Z 878.088,A -85,B 0,C 180,E1 -8540.38,E2 -8540.38} C_VEL
LIN {X 0,Y 446.423,Z 886.154,A -85,B 0,C 180,E1 -8541.399,E2 -8541.399} C_VEL
LIN {X 0,Y 446.118,Z 893.223,A -85,B 0,C 180,E1 -8542.532,E2 -8542.532} C_VEL
LIN {X 0,Y 445.968,Z 898.794,A -85,B 0,C 180,E1 -8543.667,E2 -8543.667} C_VEL
LIN {X 0,Y 445.588,Z 903.978,A -85,B 0,C 180,E1 -8545.023,E2 -8545.023} C_VEL
LIN {X 0,Y 445.622,Z 906.634,A -85,B 0,C 180,E1 -8545.93,E2 -8545.93} C_VEL
LIN {X 0,Y 445.469,Z 909.548,A -85,B 0,C 180,E1 -8547.287,E2 -8547.287} C_VEL
LIN {X 0,Y 445.379,Z 910.823,A -85,B 0,C 180,E1 -8548.191,E2 -8548.191} C_VEL
LIN {X 0,Y 445.339,Z 911.63,A -85,B 0,C 180,E1 -8549.096,E2 -8549.096} C_VEL
LIN {X 0,Y 445.34,Z 911.936,A -85,B 0,C 180,E1 -8550,E2 -8550} C_VEL
LIN {X 0,Y 445.339,Z 911.662,A -85,B 0,C 180,E1 -8550.904,E2 -8550.904} C_VEL
LIN {X 0,Y 445.379,Z 910.92,A -85,B 0,C 180,E1 -8551.809,E2 -8551.809} C_VEL
LIN {X 0,Y 445.469,Z 909.71,A -85,B 0,C 180,E1 -8552.713,E2 -8552.713} C_VEL
LIN {X 0,Y 445.619,Z 906.865,A -85,B 0,C 180,E1 -8554.07,E2 -8554.07} C_VEL
LIN {X 0,Y 445.583,Z 904.281,A -85,B 0,C 180,E1 -8554.977,E2 -8554.977} C_VEL
LIN {X 0,Y 445.945,Z 899.178,A -85,B 0,C 180,E1 -8556.334,E2 -8556.334} C_VEL
LIN {X 0,Y 446.107,Z 892.486,A -85,B 0,C 180,E1 -8557.696,E2 -8557.696} C_VEL
LIN {X 0,Y 446.48,Z 885.133,A -85,B 0,C 180,E1 -8558.828,E2 -8558.828} C_VEL
LIN {X 0,Y 446.893,Z 877.873,A -85,B 0,C 180,E1 -8559.733,E2 -8559.733} C_VEL
LIN {X 0,Y 447.22,Z 870.117,A -85,B 0,C 180,E1 -8560.526,E2 -8560.526} C_VEL
LIN {X 0,Y 447.576,Z 861.933,A -85,B 0,C 180,E1 -8561.205,E2 -8561.205} C_VEL
LIN {X 0,Y 447.828,Z 853.391,A -85,B 0,C 180,E1 -8561.772,E2 -8561.772} C_VEL
LIN {X 0,Y 448.269,Z 842.086,A -85,B 0,C 180,E1 -8562.334,E2 -8562.334} C_VEL
LIN {X 0,Y 448.455,Z 830.84,A -85,B 0,C 180,E1 -8562.692,E2 -8562.692} C_VEL
LIN {X 0,Y 448.627,Z 809.685,A -85,B 0,C 180,E1 -8563.064,E2 -8563.064} C_VEL
LIN {X 0,Y 448.784,Z 767.219,A -85,B 0,C 180,E1 -8563.744,E2 -8563.744} C_VEL
LIN {X 0,Y 446.465,Z 753.449,A -85,B 0,C 180,E1 -8564.047,E2 -8564.047} C_VEL
LIN {X 0,Y 446.98,Z 740.828,A -85,B 0,C 180,E1 -8567.382,E2 -8567.382} C_VEL
LIN {X 0,Y 446.88,Z 733.72,A -85,B 0,C 180,E1 -8569.333,E2 -8569.333} C_VEL
LIN {X 0,Y 446.546,Z 731.748,A -85,B 0,C 180,E1 -8569.958,E2 -8569.958} C_VEL
LIN {X 0,Y 446.425,Z 731.684,A -85,B 0,C 180,E1 -8573.177,E2 -8573.177} C_VEL
LIN {X 0,Y 446.434,Z 731.689,A -85,B 0,C 180,E1 -8576.191,E2 -8576.191} C_VEL
LIN {X 0,Y 446.438,Z 731.684,A -85,B 0,C 180,E1 -8579.21,E2 -8579.21} C_VEL
LIN {X 0,Y 446.421,Z 731.682,A -85,B 0,C 180,E1 -8582.362,E2 -8582.362} C_VEL
LIN {X 0,Y 446.419,Z 731.688,A -85,B 0,C 180,E1 -8585.626,E2 -8585.626} C_VEL
LIN {X 0,Y 446.427,Z 731.677,A -85,B 0,C 180,E1 -8589.029,E2 -8589.029} C_VEL
LIN {X 0,Y 446.435,Z 731.687,A -85,B 0,C 180,E1 -8592.277,E2 -8592.277} C_VEL
LIN {X 0,Y 446.452,Z 731.674,A -85,B 0,C 180,E1 -8595.104,E2 -8595.104} C_VEL
LIN {X 0,Y 446.421,Z 731.664,A -85,B 0,C 180,E1 -8598.608,E2 -8598.608} C_VEL
LIN {X 0,Y 446.443,Z 731.684,A -85,B 0,C 180,E1 -8600.973,E2 -8600.973} C_VEL
LIN {X 0,Y 446.419,Z 731.688,A -85,B 0,C 180,E1 -8604.374,E2 -8604.374} C_VEL
LIN {X 0,Y 446.421,Z 731.681,A -85,B 0,C 180,E1 -8607.638,E2 -8607.638} C_VEL
LIN {X 0,Y 446.449,Z 731.688,A -85,B 0,C 180,E1 -8610.791,E2 -8610.791} C_VEL
LIN {X 0,Y 446.48,Z 731.667,A -85,B 0,C 180,E1 -8613.848,E2 -8613.848} C_VEL
LIN {X 0,Y 446.43,Z 731.685,A -85,B 0,C 180,E1 -8616.823,E2 -8616.823} C_VEL
LIN {X 0,Y 446.446,Z 731.681,A -85,B 0,C 180,E1 -8619.737,E2 -8619.737} C_VEL
LIN {X 0,Y 446.459,Z 731.671,A -85,B 0,C 180,E1 -8622.597,E2 -8622.597} C_VEL
LIN {X 0,Y 446.474,Z 731.683,A -85,B 0,C 180,E1 -8625.412,E2 -8625.412} C_VEL
LIN {X 0,Y 446.519,Z 731.672,A -85,B 0,C 180,E1 -8628.193,E2 -8628.193} C_VEL
LIN {X 0,Y 446.602,Z 731.649,A -85,B 0,C 180,E1 -8631.858,E2 -8631.858} C_VEL
LIN {X 0,Y 446.645,Z 731.651,A -85,B 0,C 180,E1 -8634.583,E2 -8634.583} C_VEL
LIN {X 0,Y 446.711,Z 731.654,A -85,B 0,C 180,E1 -8637.295,E2 -8637.295} C_VEL
LIN {X 0,Y 446.795,Z 731.634,A -85,B 0,C 180,E1 -8640,E2 -8640} C_VEL
LIN {X 0,Y 446.693,Z 731.636,A -85,B 0,C 180,E1 -8642.705,E2 -8642.705} C_VEL
LIN {X 0,Y 446.643,Z 731.658,A -85,B 0,C 180,E1 -8646.324,E2 -8646.324} C_VEL
LIN {X 0,Y 446.54,Z 731.67,A -85,B 0,C 180,E1 -8649.055,E2 -8649.055} C_VEL
LIN {X 0,Y 446.523,Z 731.66,A -85,B 0,C 180,E1 -8652.73,E2 -8652.73} C_VEL
LIN {X 0,Y 446.498,Z 731.679,A -85,B 0,C 180,E1 -8656.228,E2 -8656.228} C_VEL
LIN {X 0,Y 446.471,Z 731.677,A -85,B 0,C 180,E1 -8659.303,E2 -8659.303} C_VEL
LIN {X 0,Y 446.421,Z 731.683,A -85,B 0,C 180,E1 -8662.199,E2 -8662.199} C_VEL
LIN {X 0,Y 446.459,Z 731.68,A -85,B 0,C 180,E1 -8665.152,E2 -8665.152} C_VEL
LIN {X 0,Y 446.486,Z 731.675,A -85,B 0,C 180,E1 -8668.178,E2 -8668.178} C_VEL
LIN {X 0,Y 446.42,Z 731.686,A -85,B 0,C 180,E1 -8671.775,E2 -8671.775} C_VEL
LIN {X 0,Y 446.432,Z 731.684,A -85,B 0,C 180,E1 -8674.523,E2 -8674.523} C_VEL
LIN {X 0,Y 446.437,Z 731.664,A -85,B 0,C 180,E1 -8678.083,E2 -8678.083} C_VEL
LIN {X 0,Y 446.444,Z 731.671,A -85,B 0,C 180,E1 -8680.92,E2 -8680.92} C_VEL
LIN {X 0,Y 446.402,Z 731.687,A -85,B 0,C 180,E1 -8683.846,E2 -8683.846} C_VEL
LIN {X 0,Y 446.416,Z 731.688,A -85,B 0,C 180,E1 -8686.401,E2 -8686.401} C_VEL
LIN {X 0,Y 446.453,Z 731.675,A -85,B 0,C 180,E1 -8689.803,E2 -8689.803} C_VEL
LIN {X 0,Y 446.43,Z 731.688,A -85,B 0,C 180,E1 -8692.123,E2 -8692.123} C_VEL
LIN {X 0,Y 446.431,Z 731.685,A -85,B 0,C 180,E1 -8695.477,E2 -8695.477} C_VEL
LIN {X 0,Y 446.417,Z 731.676,A -85,B 0,C 180,E1 -8698.7,E2 -8698.7} C_VEL
LIN {X 0,Y 446.485,Z 731.68,A -85,B 0,C 180,E1 -8701.821,E2 -8701.821} C_VEL
LIN {X 0,Y 446.496,Z 731.677,A -85,B 0,C 180,E1 -8705.347,E2 -8705.347} C_VEL
LIN {X 0,Y 446.522,Z 731.902,A -85,B 0,C 180,E1 -8705.844,E2 -8705.844} C_VEL
LIN {X 0,Y 448.048,Z 740.589,A -85,B 0,C 180,E1 -8707.885,E2 -8707.885} C_VEL
LIN {X 0,Y 447.404,Z 754.723,A -85,B 0,C 180,E1 -8710.977,E2 -8710.977} C_VEL
LIN {X 0,Y 446.773,Z 768.915,A -85,B 0,C 180,E1 -8714.05,E2 -8714.05} C_VEL
LIN {X 0,Y 446.473,Z 777.984,A -85,B 0,C 180,E1 -8715.951,E2 -8715.951} C_VEL
LIN {X 0,Y 447.318,Z 784.542,A -85,B 0,C 180,E1 -8716.121,E2 -8716.121} C_VEL
LIN {X 0,Y 448.777,Z 796.659,A -85,B 0,C 180,E1 -8716.362,E2 -8716.362} C_VEL
LIN {X 0,Y 448.403,Z 855.363,A -85,B 0,C 180,E1 -8717.325,E2 -8717.325} C_VEL
LIN {X 0,Y 448.127,Z 865.83,A -85,B 0,C 180,E1 -8717.633,E2 -8717.633} C_VEL
LIN {X 0,Y 447.804,Z 876.543,A -85,B 0,C 180,E1 -8718.113,E2 -8718.113} C_VEL
LIN {X 0,Y 447.368,Z 887.174,A -85,B 0,C 180,E1 -8718.79,E2 -8718.79} C_VEL
LIN {X 0,Y 446.997,Z 895.502,A -85,B 0,C 180,E1 -8719.468,E2 -8719.468} C_VEL
LIN {X 0,Y 446.609,Z 903.383,A -85,B 0,C 180,E1 -8720.261,E2 -8720.261} C_VEL
LIN {X 0,Y 446.256,Z 910.753,A -85,B 0,C 180,E1 -8721.167,E2 -8721.167} C_VEL
LIN {X 0,Y 445.932,Z 918.232,A -85,B 0,C 180,E1 -8722.301,E2 -8722.301} C_VEL
LIN {X 0,Y 445.664,Z 925.063,A -85,B 0,C 180,E1 -8723.662,E2 -8723.662} C_VEL
LIN {X 0,Y 445.529,Z 930.251,A -85,B 0,C 180,E1 -8725.023,E2 -8725.023} C_VEL
LIN {X 0,Y 445.433,Z 934.06,A -85,B 0,C 180,E1 -8726.382,E2 -8726.382} C_VEL
LIN {X 0,Y 445.43,Z 935.814,A -85,B 0,C 180,E1 -8727.287,E2 -8727.287} C_VEL
LIN {X 0,Y 445.351,Z 937.068,A -85,B 0,C 180,E1 -8728.191,E2 -8728.191} C_VEL
LIN {X 0,Y 445.336,Z 937.849,A -85,B 0,C 180,E1 -8729.096,E2 -8729.096} C_VEL
LIN {X 0,Y 445.339,Z 938.146,A -85,B 0,C 180,E1 -8730,E2 -8730} C_VEL
LIN {X 0,Y 445.336,Z 937.849,A -85,B 0,C 180,E1 -8730.904,E2 -8730.904} C_VEL
LIN {X 0,Y 445.351,Z 937.066,A -85,B 0,C 180,E1 -8731.809,E2 -8731.809} C_VEL
LIN {X 0,Y 445.43,Z 935.812,A -85,B 0,C 180,E1 -8732.713,E2 -8732.713} C_VEL
LIN {X 0,Y 445.436,Z 932.9,A -85,B 0,C 180,E1 -8734.071,E2 -8734.071} C_VEL
LIN {X 0,Y 445.529,Z 930.249,A -85,B 0,C 180,E1 -8734.977,E2 -8734.977} C_VEL
LIN {X 0,Y 445.664,Z 925.058,A -85,B 0,C 180,E1 -8736.338,E2 -8736.338} C_VEL
LIN {X 0,Y 445.93,Z 918.222,A -85,B 0,C 180,E1 -8737.699,E2 -8737.699} C_VEL
LIN {X 0,Y 446.255,Z 910.75,A -85,B 0,C 180,E1 -8738.833,E2 -8738.833} C_VEL
LIN {X 0,Y 446.609,Z 903.383,A -85,B 0,C 180,E1 -8739.739,E2 -8739.739} C_VEL
LIN {X 0,Y 446.997,Z 895.496,A -85,B 0,C 180,E1 -8740.532,E2 -8740.532} C_VEL
LIN {X 0,Y 447.369,Z 887.164,A -85,B 0,C 180,E1 -8741.21,E2 -8741.21} C_VEL
LIN {X 0,Y 447.868,Z 876.531,A -85,B 0,C 180,E1 -8741.886,E2 -8741.886} C_VEL
LIN {X 0,Y 448.117,Z 864.972,A -85,B 0,C 180,E1 -8742.396,E2 -8742.396} C_VEL
LIN {X 0,Y 448.417,Z 855.319,A -85,B 0,C 180,E1 -8742.675,E2 -8742.675} C_VEL
LIN {X 0,Y 448.772,Z 795.711,A -85,B 0,C 180,E1 -8743.652,E2 -8743.652} C_VEL
LIN {X 0,Y 446.468,Z 778.265,A -85,B 0,C 180,E1 -8744.026,E2 -8744.026} C_VEL
LIN {X 0,Y 446.506,Z 776.333,A -85,B 0,C 180,E1 -8744.353,E2 -8744.353} C_VEL
LIN {X 0,Y 447.107,Z 761.225,A -85,B 0,C 180,E1 -8747.613,E2 -8747.613} C_VEL
LIN {X 0,Y 447.82,Z 746.024,A -85,B 0,C 180,E1 -8750.918,E2 -8750.918} C_VEL
LIN {X 0,Y 447.974,Z 740.036,A -85,B 0,C 180,E1 -8752.239,E2 -8752.239} C_VEL
LIN {X 0,Y 446.505,Z 731.752,A -85,B 0,C 180,E1 -8754.219,E2 -8754.219} C_VEL
LIN {X 0,Y 446.479,Z 731.676,A -85,B 0,C 180,E1 -8757.161,E2 -8757.161} C_VEL
LIN {X 0,Y 446.428,Z 731.674,A -85,B 0,C 180,E1 -8760.25,E2 -8760.25} C_VEL
LIN {X 0,Y 446.445,Z 731.691,A -85,B 0,C 180,E1 -8763.454,E2 -8763.454} C_VEL
LIN {X 0,Y 446.41,Z 731.684,A -85,B 0,C 180,E1 -8766.745,E2 -8766.745} C_VEL
LIN {X 0,Y 446.484,Z 731.678,A -85,B 0,C 180,E1 -8769.53,E2 -8769.53} C_VEL
LIN {X 0,Y 446.43,Z 731.678,A -85,B 0,C 180,E1 -8772.605,E2 -8772.605} C_VEL
LIN {X 0,Y 446.454,Z 731.683,A -85,B 0,C 180,E1 -8775.103,E2 -8775.103} C_VEL
LIN {X 0,Y 446.436,Z 731.67,A -85,B 0,C 180,E1 -8778.61,E2 -8778.61} C_VEL
LIN {X 0,Y 446.471,Z 731.646,A -85,B 0,C 180,E1 -8780.976,E2 -8780.976} C_VEL
LIN {X 0,Y 446.423,Z 731.683,A -85,B 0,C 180,E1 -8784.374,E2 -8784.374} C_VEL
LIN {X 0,Y 446.423,Z 731.69,A -85,B 0,C 180,E1 -8787.639,E2 -8787.639} C_VEL
LIN {X 0,Y 446.45,Z 731.673,A -85,B 0,C 180,E1 -8790.791,E2 -8790.791} C_VEL
LIN {X 0,Y 446.479,Z 731.683,A -85,B 0,C 180,E1 -8793.849,E2 -8793.849} C_VEL
LIN {X 0,Y 446.431,Z 731.679,A -85,B 0,C 180,E1 -8796.824,E2 -8796.824} C_VEL
LIN {X 0,Y 446.447,Z 731.674,A -85,B 0,C 180,E1 -8799.737,E2 -8799.737} C_VEL
LIN {X 0,Y 446.466,Z 731.682,A -85,B 0,C 180,E1 -8802.597,E2 -8802.597} C_VEL
LIN {X 0,Y 446.472,Z 731.675,A -85,B 0,C 180,E1 -8805.413,E2 -8805.413} C_VEL
LIN {X 0,Y 446.519,Z 731.664,A -85,B 0,C 180,E1 -8808.193,E2 -8808.193} C_VEL
LIN {X 0,Y 446.602,Z 731.664,A -85,B 0,C 180,E1 -8811.858,E2 -8811.858} C_VEL
LIN {X 0,Y 446.645,Z 731.658,A -85,B 0,C 180,E1 -8814.583,E2 -8814.583} C_VEL
LIN {X 0,Y 446.666,Z 731.643,A -85,B 0,C 180,E1 -8818.197,E2 -8818.197} C_VEL
LIN {X 0,Y 446.796,Z 731.633,A -85,B 0,C 180,E1 -8820,E2 -8820} C_VEL
LIN {X 0,Y 446.711,Z 731.654,A -85,B 0,C 180,E1 -8822.705,E2 -8822.705} C_VEL
LIN {X 0,Y 446.641,Z 731.655,A -85,B 0,C 180,E1 -8826.324,E2 -8826.324} C_VEL
LIN {X 0,Y 446.539,Z 731.669,A -85,B 0,C 180,E1 -8829.055,E2 -8829.055} C_VEL
LIN {X 0,Y 446.523,Z 731.68,A -85,B 0,C 180,E1 -8832.73,E2 -8832.73} C_VEL
LIN {X 0,Y 446.497,Z 731.669,A -85,B 0,C 180,E1 -8836.228,E2 -8836.228} C_VEL
LIN {X 0,Y 446.47,Z 731.68,A -85,B 0,C 180,E1 -8839.303,E2 -8839.303} C_VEL
LIN {X 0,Y 446.419,Z 731.686,A -85,B 0,C 180,E1 -8842.2,E2 -8842.2} C_VEL
LIN {X 0,Y 446.448,Z 731.676,A -85,B 0,C 180,E1 -8845.153,E2 -8845.153} C_VEL
LIN {X 0,Y 446.486,Z 731.675,A -85,B 0,C 180,E1 -8848.179,E2 -8848.179} C_VEL
LIN {X 0,Y 446.419,Z 731.682,A -85,B 0,C 180,E1 -8851.775,E2 -8851.775} C_VEL
LIN {X 0,Y 446.424,Z 731.68,A -85,B 0,C 180,E1 -8854.524,E2 -8854.524} C_VEL
LIN {X 0,Y 446.416,Z 731.685,A -85,B 0,C 180,E1 -8858.079,E2 -8858.079} C_VEL
LIN {X 0,Y 446.425,Z 731.676,A -85,B 0,C 180,E1 -8860.917,E2 -8860.917} C_VEL
LIN {X 0,Y 446.4,Z 731.676,A -85,B 0,C 180,E1 -8863.846,E2 -8863.846} C_VEL
LIN {X 0,Y 446.397,Z 731.687,A -85,B 0,C 180,E1 -8866.404,E2 -8866.404} C_VEL
LIN {X 0,Y 446.428,Z 731.687,A -85,B 0,C 180,E1 -8869.082,E2 -8869.082} C_VEL
LIN {X 0,Y 446.409,Z 731.68,A -85,B 0,C 180,E1 -8872.121,E2 -8872.121} C_VEL
LIN {X 0,Y 446.425,Z 731.693,A -85,B 0,C 180,E1 -8875.477,E2 -8875.477} C_VEL
LIN {X 0,Y 446.416,Z 731.679,A -85,B 0,C 180,E1 -8878.7,E2 -8878.7} C_VEL
LIN {X 0,Y 446.451,Z 731.686,A -85,B 0,C 180,E1 -8881.83,E2 -8881.83} C_VEL
LIN {X 0,Y 446.44,Z 731.684,A -85,B 0,C 180,E1 -8884.847,E2 -8884.847} C_VEL
LIN {X 0,Y 446.45,Z 731.685,A -85,B 0,C 180,E1 -8888.245,E2 -8888.245} C_VEL
LIN {X 0,Y 446.558,Z 731.859,A -85,B 0,C 180,E1 -8890.223,E2 -8890.223} C_VEL
LIN {X 0,Y 447.074,Z 737.021,A -85,B 0,C 180,E1 -8891.675,E2 -8891.675} C_VEL
LIN {X 0,Y 446.705,Z 747.519,A -85,B 0,C 180,E1 -8894.487,E2 -8894.487} C_VEL
LIN {X 0,Y 446.497,Z 753.636,A -85,B 0,C 180,E1 -8896.017,E2 -8896.017} C_VEL
LIN {X 0,Y 447.689,Z 760.66,A -85,B 0,C 180,E1 -8896.207,E2 -8896.207} C_VEL
LIN {X 0,Y 448.912,Z 768.122,A -85,B 0,C 180,E1 -8896.366,E2 -8896.366} C_VEL
LIN {X 0,Y 448.638,Z 812.291,A -85,B 0,C 180,E1 -8897.07,E2 -8897.07} C_VEL
LIN {X 0,Y 447.937,Z 818.14,A -85,B 0,C 180,E1 -8897.141,E2 -8897.141} C_VEL
LIN {X 0,Y 443.148,Z 833.228,A -85,B 0,C 180,E1 -8897.298,E2 -8897.298} C_VEL
LIN {X 0,Y 441.464,Z 840.77,A -85,B 0,C 180,E1 -8897.505,E2 -8897.505} C_VEL
LIN {X 0,Y 441.325,Z 842.656,A -85,B 0,C 180,E1 -8897.577,E2 -8897.577} C_VEL
LIN {X 0,Y 440.948,Z 852.126,A -85,B 0,C 180,E1 -8898.042,E2 -8898.042} C_VEL
LIN {X 0,Y 440.686,Z 860.958,A -85,B 0,C 180,E1 -8898.618,E2 -8898.618} C_VEL
LIN {X 0,Y 440.262,Z 869.358,A -85,B 0,C 180,E1 -8899.305,E2 -8899.305} C_VEL
LIN {X 0,Y 439.913,Z 877.283,A -85,B 0,C 180,E1 -8900.111,E2 -8900.111} C_VEL
LIN {X 0,Y 439.565,Z 882.976,A -85,B 0,C 180,E1 -8900.8,E2 -8900.8} C_VEL
LIN {X 0,Y 439.259,Z 889.326,A -85,B 0,C 180,E1 -8901.721,E2 -8901.721} C_VEL
LIN {X 0,Y 438.975,Z 895.739,A -85,B 0,C 180,E1 -8902.866,E2 -8902.866} C_VEL
LIN {X 0,Y 438.92,Z 899.005,A -85,B 0,C 180,E1 -8903.565,E2 -8903.565} C_VEL
LIN {X 0,Y 438.526,Z 904.188,A -85,B 0,C 180,E1 -8904.943,E2 -8904.943} C_VEL
LIN {X 0,Y 438.539,Z 906.844,A -85,B 0,C 180,E1 -8905.864,E2 -8905.864} C_VEL
LIN {X 0,Y 438.401,Z 909.757,A -85,B 0,C 180,E1 -8907.243,E2 -8907.243} C_VEL
LIN {X 0,Y 438.3,Z 911.032,A -85,B 0,C 180,E1 -8908.162,E2 -8908.162} C_VEL
LIN {X 0,Y 438.253,Z 911.839,A -85,B 0,C 180,E1 -8909.081,E2 -8909.081} C_VEL
LIN {X 0,Y 438.252,Z 912.145,A -85,B 0,C 180,E1 -8910,E2 -8910} C_VEL
LIN {X 0,Y 438.253,Z 911.87,A -85,B 0,C 180,E1 -8910.919,E2 -8910.919} C_VEL
LIN {X 0,Y 438.301,Z 911.128,A -85,B 0,C 180,E1 -8911.838,E2 -8911.838} C_VEL
LIN {X 0,Y 438.401,Z 909.917,A -85,B 0,C 180,E1 -8912.757,E2 -8912.757} C_VEL
LIN {X 0,Y 438.535,Z 907.072,A -85,B 0,C 180,E1 -8914.136,E2 -8914.136} C_VEL
LIN {X 0,Y 438.521,Z 904.488,A -85,B 0,C 180,E1 -8915.057,E2 -8915.057} C_VEL
LIN {X 0,Y 438.898,Z 899.385,A -85,B 0,C 180,E1 -8916.436,E2 -8916.436} C_VEL
LIN {X 0,Y 439.01,Z 893.904,A -85,B 0,C 180,E1 -8917.589,E2 -8917.589} C_VEL
LIN {X 0,Y 439.369,Z 887.013,A -85,B 0,C 180,E1 -8918.74,E2 -8918.74} C_VEL
LIN {X 0,Y 439.832,Z 879.096,A -85,B 0,C 180,E1 -8919.775,E2 -8919.775} C_VEL
LIN {X 0,Y 440.155,Z 871.547,A -85,B 0,C 180,E1 -8920.581,E2 -8920.581} C_VEL
LIN {X 0,Y 440.533,Z 863.633,A -85,B 0,C 180,E1 -8921.27,E2 -8921.27} C_VEL
LIN {X 0,Y 440.874,Z 855.46,A -85,B 0,C 180,E1 -8921.844,E2 -8921.844} C_VEL
LIN {X 0,Y 441.221,Z 847.18,A -85,B 0,C 180,E1 -8922.301,E2 -8922.301} C_VEL
LIN {X 0,Y 441.443,Z 838.242,A -85,B 0,C 180,E1 -8922.674,E2 -8922.674} C_VEL
LIN {X 0,Y 441.636,Z 828.717,A -85,B 0,C 180,E1 -8922.943,E2 -8922.943} C_VEL
LIN {X 0,Y 441.937,Z 768.164,A -85,B 0,C 180,E1 -8923.948,E2 -8923.948} C_VEL
LIN {X 0,Y 439.478,Z 753.578,A -85,B 0,C 180,E1 -8924.292,E2 -8924.292} C_VEL
LIN {X 0,Y 440,Z 741.005,A -85,B 0,C 180,E1 -8927.667,E2 -8927.667} C_VEL
LIN {X 0,Y 439.813,Z 734.531,A -85,B 0,C 180,E1 -8929.474,E2 -8929.474} C_VEL
LIN {X 0,Y 439.481,Z 732.617,A -85,B 0,C 180,E1 -8930.11,E2 -8930.11} C_VEL
LIN {X 0,Y 439.383,Z 732.561,A -85,B 0,C 180,E1 -8933.571,E2 -8933.571} C_VEL
LIN {X 0,Y 439.38,Z 732.567,A -85,B 0,C 180,E1 -8936.607,E2 -8936.607} C_VEL
LIN {X 0,Y 439.378,Z 732.565,A -85,B 0,C 180,E1 -8939.726,E2 -8939.726} C_VEL
LIN {X 0,Y 439.373,Z 732.564,A -85,B 0,C 180,E1 -8942.946,E2 -8942.946} C_VEL
LIN {X 0,Y 439.374,Z 732.568,A -85,B 0,C 180,E1 -8946.287,E2 -8946.287} C_VEL
LIN {X 0,Y 439.403,Z 732.551,A -85,B 0,C 180,E1 -8949.849,E2 -8949.849} C_VEL
LIN {X 0,Y 439.383,Z 732.569,A -85,B 0,C 180,E1 -8952.627,E2 -8952.627} C_VEL
LIN {X 0,Y 439.4,Z 732.55,A -85,B 0,C 180,E1 -8955.27,E2 -8955.27} C_VEL
LIN {X 0,Y 439.383,Z 732.542,A -85,B 0,C 180,E1 -8958.744,E2 -8958.744} C_VEL
LIN {X 0,Y 439.374,Z 732.561,A -85,B 0,C 180,E1 -8961.608,E2 -8961.608} C_VEL
LIN {X 0,Y 439.398,Z 732.563,A -85,B 0,C 180,E1 -8964.844,E2 -8964.844} C_VEL
LIN {X 0,Y 439.373,Z 732.559,A -85,B 0,C 180,E1 -8968.139,E2 -8968.139} C_VEL
LIN {X 0,Y 439.434,Z 732.554,A -85,B 0,C 180,E1 -8971.598,E2 -8971.598} C_VEL
LIN {X 0,Y 439.402,Z 732.549,A -85,B 0,C 180,E1 -8974.415,E2 -8974.415} C_VEL
LIN {X 0,Y 439.366,Z 732.567,A -85,B 0,C 180,E1 -8977.425,E2 -8977.425} C_VEL
LIN {X 0,Y 439.443,Z 732.554,A -85,B 0,C 180,E1 -8980.663,E2 -8980.663} C_VEL
LIN {X 0,Y 439.465,Z 732.544,A -85,B 0,C 180,E1 -8984.224,E2 -8984.224} C_VEL
LIN {X 0,Y 439.485,Z 732.549,A -85,B 0,C 180,E1 -8988.001,E2 -8988.001} C_VEL
LIN {X 0,Y 439.55,Z 732.528,A -85,B 0,C 180,E1 -8991.726,E2 -8991.726} C_VEL
LIN {X 0,Y 439.62,Z 732.526,A -85,B 0,C 180,E1 -8994.496,E2 -8994.496} C_VEL
LIN {X 0,Y 439.638,Z 732.53,A -85,B 0,C 180,E1 -8998.168,E2 -8998.168} C_VEL
LIN {X 0,Y 439.764,Z 732.509,A -85,B 0,C 180,E1 -9000,E2 -9000} C_VEL
LIN {X 0,Y 439.643,Z 732.514,A -85,B 0,C 180,E1 -9002.749,E2 -9002.749} C_VEL
LIN {X 0,Y 439.615,Z 732.533,A -85,B 0,C 180,E1 -9006.425,E2 -9006.425} C_VEL
LIN {X 0,Y 439.502,Z 732.548,A -85,B 0,C 180,E1 -9009.201,E2 -9009.201} C_VEL
LIN {X 0,Y 439.467,Z 732.539,A -85,B 0,C 180,E1 -9012.937,E2 -9012.937} C_VEL
LIN {X 0,Y 439.449,Z 732.555,A -85,B 0,C 180,E1 -9016.349,E2 -9016.349} C_VEL
LIN {X 0,Y 439.433,Z 732.557,A -85,B 0,C 180,E1 -9019.625,E2 -9019.625} C_VEL
LIN {X 0,Y 439.367,Z 732.56,A -85,B 0,C 180,E1 -9022.575,E2 -9022.575} C_VEL
LIN {X 0,Y 439.407,Z 732.561,A -85,B 0,C 180,E1 -9025.585,E2 -9025.585} C_VEL
LIN {X 0,Y 439.419,Z 732.549,A -85,B 0,C 180,E1 -9028.673,E2 -9028.673} C_VEL
LIN {X 0,Y 439.371,Z 732.567,A -85,B 0,C 180,E1 -9032.03,E2 -9032.03} C_VEL
LIN {X 0,Y 439.398,Z 732.556,A -85,B 0,C 180,E1 -9035.341,E2 -9035.341} C_VEL
LIN {X 0,Y 439.396,Z 732.531,A -85,B 0,C 180,E1 -9038.593,E2 -9038.593} C_VEL
LIN {X 0,Y 439.399,Z 732.547,A -85,B 0,C 180,E1 -9041.258,E2 -9041.258} C_VEL
LIN {X 0,Y 439.402,Z 732.564,A -85,B 0,C 180,E1 -9044.729,E2 -9044.729} C_VEL
LIN {X 0,Y 439.396,Z 732.554,A -85,B 0,C 180,E1 -9047.796,E2 -9047.796} C_VEL
LIN {X 0,Y 439.441,Z 732.552,A -85,B 0,C 180,E1 -9050.229,E2 -9050.229} C_VEL
LIN {X 0,Y 439.378,Z 732.558,A -85,B 0,C 180,E1 -9053.713,E2 -9053.713} C_VEL
LIN {X 0,Y 439.373,Z 732.564,A -85,B 0,C 180,E1 -9057.054,E2 -9057.054} C_VEL
LIN {X 0,Y 439.383,Z 732.555,A -85,B 0,C 180,E1 -9060.274,E2 -9060.274} C_VEL
LIN {X 0,Y 439.43,Z 732.551,A -85,B 0,C 180,E1 -9063.396,E2 -9063.396} C_VEL
LIN {X 0,Y 439.495,Z 732.66,A -85,B 0,C 180,E1 -9065.627,E2 -9065.627} C_VEL
LIN {X 0,Y 440.919,Z 740.78,A -85,B 0,C 180,E1 -9067.591,E2 -9067.591} C_VEL
LIN {X 0,Y 440.888,Z 745.854,A -85,B 0,C 180,E1 -9068.737,E2 -9068.737} C_VEL
LIN {X 0,Y 440.122,Z 761.038,A -85,B 0,C 180,E1 -9072.098,E2 -9072.098} C_VEL
LIN {X 0,Y 439.519,Z 775.058,A -85,B 0,C 180,E1 -9075.176,E2 -9075.176} C_VEL
LIN {X 0,Y 439.444,Z 777.782,A -85,B 0,C 180,E1 -9075.721,E2 -9075.721} C_VEL
LIN {X 0,Y 440.233,Z 783.916,A -85,B 0,C 180,E1 -9075.886,E2 -9075.886} C_VEL
LIN {X 0,Y 441.892,Z 798.074,A -85,B 0,C 180,E1 -9076.172,E2 -9076.172} C_VEL
LIN {X 0,Y 441.486,Z 855.165,A -85,B 0,C 180,E1 -9077.123,E2 -9077.123} C_VEL
LIN {X 0,Y 441.202,Z 865.628,A -85,B 0,C 180,E1 -9077.436,E2 -9077.436} C_VEL
LIN {X 0,Y 440.861,Z 876.339,A -85,B 0,C 180,E1 -9077.923,E2 -9077.923} C_VEL
LIN {X 0,Y 440.406,Z 886.969,A -85,B 0,C 180,E1 -9078.61,E2 -9078.61} C_VEL
LIN {X 0,Y 440.011,Z 895.295,A -85,B 0,C 180,E1 -9079.299,E2 -9079.299} C_VEL
LIN {X 0,Y 439.609,Z 903.176,A -85,B 0,C 180,E1 -9080.104,E2 -9080.104} C_VEL
LIN {X 0,Y 439.237,Z 910.546,A -85,B 0,C 180,E1 -9081.025,E2 -9081.025} C_VEL
LIN {X 0,Y 438.886,Z 918.024,A -85,B 0,C 180,E1 -9082.177,E2 -9082.177} C_VEL
LIN {X 0,Y 438.592,Z 924.855,A -85,B 0,C 180,E1 -9083.56,E2 -9083.56} C_VEL
LIN {X 0,Y 438.462,Z 930.043,A -85,B 0,C 180,E1 -9084.942,E2 -9084.942} C_VEL
LIN {X 0,Y 438.333,Z 933.851,A -85,B 0,C 180,E1 -9086.323,E2 -9086.323} C_VEL
LIN {X 0,Y 438.341,Z 935.605,A -85,B 0,C 180,E1 -9087.243,E2 -9087.243} C_VEL
LIN {X 0,Y 438.274,Z 936.859,A -85,B 0,C 180,E1 -9088.162,E2 -9088.162} C_VEL
LIN {X 0,Y 438.249,Z 937.641,A -85,B 0,C 180,E1 -9089.081,E2 -9089.081} C_VEL
LIN {X 0,Y 438.25,Z 937.937,A -85,B 0,C 180,E1 -9090,E2 -9090} C_VEL
LIN {X 0,Y 438.249,Z 937.64,A -85,B 0,C 180,E1 -9090.919,E2 -9090.919} C_VEL
LIN {X 0,Y 438.274,Z 936.858,A -85,B 0,C 180,E1 -9091.838,E2 -9091.838} C_VEL
LIN {X 0,Y 438.341,Z 935.602,A -85,B 0,C 180,E1 -9092.757,E2 -9092.757} C_VEL
LIN {X 0,Y 438.347,Z 932.69,A -85,B 0,C 180,E1 -9094.137,E2 -9094.137} C_VEL
LIN {X 0,Y 438.462,Z 930.039,A -85,B 0,C 180,E1 -9095.058,E2 -9095.058} C_VEL
LIN {X 0,Y 438.592,Z 924.848,A -85,B 0,C 180,E1 -9096.44,E2 -9096.44} C_VEL
LIN {X 0,Y 438.885,Z 918.012,A -85,B 0,C 180,E1 -9097.823,E2 -9097.823} C_VEL
LIN {X 0,Y 439.221,Z 910.539,A -85,B 0,C 180,E1 -9098.975,E2 -9098.975} C_VEL
LIN {X 0,Y 439.609,Z 903.171,A -85,B 0,C 180,E1 -9099.896,E2 -9099.896} C_VEL
LIN {X 0,Y 440.011,Z 895.284,A -85,B 0,C 180,E1 -9100.701,E2 -9100.701} C_VEL
LIN {X 0,Y 440.397,Z 886.951,A -85,B 0,C 180,E1 -9101.39,E2 -9101.39} C_VEL
LIN {X 0,Y 440.827,Z 878.23,A -85,B 0,C 180,E1 -9101.962,E2 -9101.962} C_VEL
LIN {X 0,Y 441.139,Z 866.421,A -85,B 0,C 180,E1 -9102.537,E2 -9102.537} C_VEL
LIN {X 0,Y 441.474,Z 856.397,A -85,B 0,C 180,E1 -9102.849,E2 -9102.849} C_VEL
LIN {X 0,Y 441.667,Z 832.99,A -85,B 0,C 180,E1 -9103.262,E2 -9103.262} C_VEL
LIN {X 0,Y 441.734,Z 794.843,A -85,B 0,C 180,E1 -9103.884,E2 -9103.884} C_VEL
LIN {X 0,Y 439.47,Z 778.181,A -85,B 0,C 180,E1 -9104.246,E2 -9104.246} C_VEL
LIN {X 0,Y 439.503,Z 776.238,A -85,B 0,C 180,E1 -9104.564,E2 -9104.564} C_VEL
LIN {X 0,Y 440.073,Z 762.122,A -85,B 0,C 180,E1 -9107.664,E2 -9107.664} C_VEL
LIN {X 0,Y 440.825,Z 746.937,A -85,B 0,C 180,E1 -9111.021,E2 -9111.021} C_VEL
LIN {X 0,Y 441.021,Z 741.337,A -85,B 0,C 180,E1 -9112.276,E2 -9112.276} C_VEL
LIN {X 0,Y 439.495,Z 732.613,A -85,B 0,C 180,E1 -9114.397,E2 -9114.397} C_VEL
LIN {X 0,Y 439.443,Z 732.558,A -85,B 0,C 180,E1 -9117.632,E2 -9117.632} C_VEL
LIN {X 0,Y 439.362,Z 732.552,A -85,B 0,C 180,E1 -9120.788,E2 -9120.788} C_VEL
LIN {X 0,Y 439.388,Z 732.564,A -85,B 0,C 180,E1 -9124.044,E2 -9124.044} C_VEL
LIN {X 0,Y 439.358,Z 732.563,A -85,B 0,C 180,E1 -9126.889,E2 -9126.889} C_VEL
LIN {X 0,Y 439.417,Z 732.554,A -85,B 0,C 180,E1 -9129.852,E2 -9129.852} C_VEL
LIN {X 0,Y 439.383,Z 732.555,A -85,B 0,C 180,E1 -9132.627,E2 -9132.627} C_VEL
LIN {X 0,Y 439.402,Z 732.563,A -85,B 0,C 180,E1 -9135.271,E2 -9135.271} C_VEL
LIN {X 0,Y 439.399,Z 732.546,A -85,B 0,C 180,E1 -9138.742,E2 -9138.742} C_VEL
LIN {X 0,Y 439.391,Z 732.534,A -85,B 0,C 180,E1 -9141.605,E2 -9141.605} C_VEL
LIN {X 0,Y 439.402,Z 732.556,A -85,B 0,C 180,E1 -9144.844,E2 -9144.844} C_VEL
LIN {X 0,Y 439.374,Z 732.564,A -85,B 0,C 180,E1 -9148.14,E2 -9148.14} C_VEL
LIN {X 0,Y 439.433,Z 732.55,A -85,B 0,C 180,E1 -9151.598,E2 -9151.598} C_VEL
LIN {X 0,Y 439.407,Z 732.561,A -85,B 0,C 180,E1 -9154.415,E2 -9154.415} C_VEL
LIN {X 0,Y 439.367,Z 732.559,A -85,B 0,C 180,E1 -9157.425,E2 -9157.425} C_VEL
LIN {X 0,Y 439.443,Z 732.553,A -85,B 0,C 180,E1 -9160.663,E2 -9160.663} C_VEL
LIN {X 0,Y 439.464,Z 732.556,A -85,B 0,C 180,E1 -9164.225,E2 -9164.225} C_VEL
LIN {X 0,Y 439.485,Z 732.539,A -85,B 0,C 180,E1 -9168.001,E2 -9168.001} C_VEL
LIN {X 0,Y 439.55,Z 732.541,A -85,B 0,C 180,E1 -9171.726,E2 -9171.726} C_VEL
LIN {X 0,Y 439.621,Z 732.534,A -85,B 0,C 180,E1 -9174.496,E2 -9174.496} C_VEL
LIN {X 0,Y 439.636,Z 732.517,A -85,B 0,C 180,E1 -9178.168,E2 -9178.168} C_VEL
LIN {X 0,Y 439.766,Z 732.509,A -85,B 0,C 180,E1 -9180,E2 -9180} C_VEL
LIN {X 0,Y 439.658,Z 732.532,A -85,B 0,C 180,E1 -9182.749,E2 -9182.749} C_VEL
LIN {X 0,Y 439.616,Z 732.528,A -85,B 0,C 180,E1 -9186.425,E2 -9186.425} C_VEL
LIN {X 0,Y 439.501,Z 732.544,A -85,B 0,C 180,E1 -9189.202,E2 -9189.202} C_VEL
LIN {X 0,Y 439.467,Z 732.556,A -85,B 0,C 180,E1 -9192.938,E2 -9192.938} C_VEL
LIN {X 0,Y 439.448,Z 732.548,A -85,B 0,C 180,E1 -9196.348,E2 -9196.348} C_VEL
LIN {X 0,Y 439.404,Z 732.557,A -85,B 0,C 180,E1 -9199.626,E2 -9199.626} C_VEL
LIN {X 0,Y 439.366,Z 732.567,A -85,B 0,C 180,E1 -9202.575,E2 -9202.575} C_VEL
LIN {X 0,Y 439.401,Z 732.549,A -85,B 0,C 180,E1 -9205.585,E2 -9205.585} C_VEL
LIN {X 0,Y 439.419,Z 732.558,A -85,B 0,C 180,E1 -9208.673,E2 -9208.673} C_VEL
LIN {X 0,Y 439.369,Z 732.559,A -85,B 0,C 180,E1 -9212.03,E2 -9212.03} C_VEL
LIN {X 0,Y 439.393,Z 732.565,A -85,B 0,C 180,E1 -9215.34,E2 -9215.34} C_VEL
LIN {X 0,Y 439.378,Z 732.562,A -85,B 0,C 180,E1 -9218.596,E2 -9218.596} C_VEL
LIN {X 0,Y 439.383,Z 732.544,A -85,B 0,C 180,E1 -9221.256,E2 -9221.256} C_VEL
LIN {X 0,Y 439.4,Z 732.549,A -85,B 0,C 180,E1 -9224.73,E2 -9224.73} C_VEL
LIN {X 0,Y 439.397,Z 732.564,A -85,B 0,C 180,E1 -9227.796,E2 -9227.796} C_VEL
LIN {X 0,Y 439.396,Z 732.552,A -85,B 0,C 180,E1 -9230.224,E2 -9230.224} C_VEL
LIN {X 0,Y 439.374,Z 732.566,A -85,B 0,C 180,E1 -9233.713,E2 -9233.713} C_VEL
LIN {X 0,Y 439.373,Z 732.564,A -85,B 0,C 180,E1 -9237.054,E2 -9237.054} C_VEL
LIN {X 0,Y 439.378,Z 732.566,A -85,B 0,C 180,E1 -9240.274,E2 -9240.274} C_VEL
LIN {X 0,Y 439.383,Z 732.566,A -85,B 0,C 180,E1 -9243.393,E2 -9243.393} C_VEL
LIN {X 0,Y 439.383,Z 732.561,A -85,B 0,C 180,E1 -9246.429,E2 -9246.429} C_VEL
LIN {X 0,Y 439.458,Z 732.569,A -85,B 0,C 180,E1 -9249.889,E2 -9249.889} C_VEL
LIN {X 0,Y 439.531,Z 732.87,A -85,B 0,C 180,E1 -9250.136,E2 -9250.136} C_VEL
LIN {X 0,Y 440.054,Z 737.193,A -85,B 0,C 180,E1 -9251.372,E2 -9251.372} C_VEL
LIN {X 0,Y 439.727,Z 747.709,A -85,B 0,C 180,E1 -9254.234,E2 -9254.234} C_VEL
LIN {X 0,Y 439.46,Z 753.781,A -85,B 0,C 180,E1 -9255.783,E2 -9255.783} C_VEL
LIN {X 0,Y 440.322,Z 758.612,A -85,B 0,C 180,E1 -9255.933,E2 -9255.933} C_VEL
LIN {X 0,Y 442.013,Z 768.683,A -85,B 0,C 180,E1 -9256.154,E2 -9256.154} C_VEL
LIN {X 0,Y 441.577,Z 829.066,A -85,B 0,C 180,E1 -9257.155,E2 -9257.155} C_VEL
LIN {X 0,Y 441.426,Z 838.96,A -85,B 0,C 180,E1 -9257.442,E2 -9257.442} C_VEL
LIN {X 0,Y 441.325,Z 842.656,A -85,B 0,C 180,E1 -9257.577,E2 -9257.577} C_VEL
LIN {X 0,Y 440.535,Z 846.427,A -85,B 0,C 180,E1 -9257.719,E2 -9257.719} C_VEL
LIN {X 0,Y 437.547,Z 852.28,A -85,B 0,C 180,E1 -9257.937,E2 -9257.937} C_VEL
LIN {X 0,Y 434.548,Z 857.957,A -85,B 0,C 180,E1 -9258.215,E2 -9258.215} C_VEL
LIN {X 0,Y 433.737,Z 861.404,A -85,B 0,C 180,E1 -9258.451,E2 -9258.451} C_VEL
LIN {X 0,Y 433.287,Z 869.572,A -85,B 0,C 180,E1 -9259.131,E2 -9259.131} C_VEL
LIN {X 0,Y 432.918,Z 877.496,A -85,B 0,C 180,E1 -9259.95,E2 -9259.95} C_VEL
LIN {X 0,Y 432.571,Z 883.188,A -85,B 0,C 180,E1 -9260.65,E2 -9260.65} C_VEL
LIN {X 0,Y 432.226,Z 889.538,A -85,B 0,C 180,E1 -9261.585,E2 -9261.585} C_VEL
LIN {X 0,Y 431.966,Z 894.814,A -85,B 0,C 180,E1 -9262.521,E2 -9262.521} C_VEL
LIN {X 0,Y 431.88,Z 899.216,A -85,B 0,C 180,E1 -9263.459,E2 -9263.459} C_VEL
LIN {X 0,Y 431.47,Z 904.398,A -85,B 0,C 180,E1 -9264.86,E2 -9264.86} C_VEL
LIN {X 0,Y 431.44,Z 907.055,A -85,B 0,C 180,E1 -9265.796,E2 -9265.796} C_VEL
LIN {X 0,Y 431.334,Z 909.966,A -85,B 0,C 180,E1 -9267.198,E2 -9267.198} C_VEL
LIN {X 0,Y 431.225,Z 911.241,A -85,B 0,C 180,E1 -9268.132,E2 -9268.132} C_VEL
LIN {X 0,Y 431.17,Z 912.047,A -85,B 0,C 180,E1 -9269.066,E2 -9269.066} C_VEL
LIN {X 0,Y 431.166,Z 912.354,A -85,B 0,C 180,E1 -9270,E2 -9270} C_VEL
LIN {X 0,Y 431.17,Z 912.079,A -85,B 0,C 180,E1 -9270.934,E2 -9270.934} C_VEL
LIN {X 0,Y 431.225,Z 911.336,A -85,B 0,C 180,E1 -9271.868,E2 -9271.868} C_VEL
LIN {X 0,Y 431.334,Z 910.125,A -85,B 0,C 180,E1 -9272.802,E2 -9272.802} C_VEL
LIN {X 0,Y 431.436,Z 907.28,A -85,B 0,C 180,E1 -9274.204,E2 -9274.204} C_VEL
LIN {X 0,Y 431.465,Z 904.694,A -85,B 0,C 180,E1 -9275.14,E2 -9275.14} C_VEL
LIN {X 0,Y 431.829,Z 899.592,A -85,B 0,C 180,E1 -9276.542,E2 -9276.542} C_VEL
LIN {X 0,Y 431.962,Z 894.11,A -85,B 0,C 180,E1 -9277.714,E2 -9277.714} C_VEL
LIN {X 0,Y 432.367,Z 887.218,A -85,B 0,C 180,E1 -9278.883,E2 -9278.883} C_VEL
LIN {X 0,Y 432.85,Z 879.3,A -85,B 0,C 180,E1 -9279.934,E2 -9279.934} C_VEL
LIN {X 0,Y 433.193,Z 871.75,A -85,B 0,C 180,E1 -9280.753,E2 -9280.753} C_VEL
LIN {X 0,Y 433.574,Z 863.836,A -85,B 0,C 180,E1 -9281.453,E2 -9281.453} C_VEL
LIN {X 0,Y 433.923,Z 855.662,A -85,B 0,C 180,E1 -9282.036,E2 -9282.036} C_VEL
LIN {X 0,Y 434.297,Z 847.379,A -85,B 0,C 180,E1 -9282.5,E2 -9282.5} C_VEL
LIN {X 0,Y 434.54,Z 838.436,A -85,B 0,C 180,E1 -9282.879,E2 -9282.879} C_VEL
LIN {X 0,Y 434.701,Z 829.005,A -85,B 0,C 180,E1 -9283.151,E2 -9283.151} C_VEL
LIN {X 0,Y 435.036,Z 768.666,A -85,B 0,C 180,E1 -9284.169,E2 -9284.169} C_VEL
LIN {X 0,Y 432.445,Z 753.778,A -85,B 0,C 180,E1 -9284.53,E2 -9284.53} C_VEL
LIN {X 0,Y 432.942,Z 742.941,A -85,B 0,C 180,E1 -9287.476,E2 -9287.476} C_VEL
LIN {X 0,Y 432.922,Z 736.491,A -85,B 0,C 180,E1 -9289.283,E2 -9289.283} C_VEL
LIN {X 0,Y 432.442,Z 733.518,A -85,B 0,C 180,E1 -9290.203,E2 -9290.203} C_VEL
LIN {X 0,Y 432.366,Z 733.437,A -85,B 0,C 180,E1 -9293.977,E2 -9293.977} C_VEL
LIN {X 0,Y 432.322,Z 733.443,A -85,B 0,C 180,E1 -9297.076,E2 -9297.076} C_VEL
LIN {X 0,Y 432.345,Z 733.442,A -85,B 0,C 180,E1 -9300.26,E2 -9300.26} C_VEL
LIN {X 0,Y 432.34,Z 733.439,A -85,B 0,C 180,E1 -9303.552,E2 -9303.552} C_VEL
LIN {X 0,Y 432.338,Z 733.443,A -85,B 0,C 180,E1 -9305.818,E2 -9305.818} C_VEL
LIN {X 0,Y 432.323,Z 733.432,A -85,B 0,C 180,E1 -9309.346,E2 -9309.346} C_VEL
LIN {X 0,Y 432.334,Z 733.44,A -85,B 0,C 180,E1 -9311.797,E2 -9311.797} C_VEL
LIN {X 0,Y 432.335,Z 733.443,A -85,B 0,C 180,E1 -9314.347,E2 -9314.347} C_VEL
LIN {X 0,Y 432.317,Z 733.414,A -85,B 0,C 180,E1 -9317.016,E2 -9317.016} C_VEL
LIN {X 0,Y 432.333,Z 733.428,A -85,B 0,C 180,E1 -9319.821,E2 -9319.821} C_VEL
LIN {X 0,Y 432.308,Z 733.448,A -85,B 0,C 180,E1 -9323.022,E2 -9323.022} C_VEL
LIN {X 0,Y 432.359,Z 733.431,A -85,B 0,C 180,E1 -9325.997,E2 -9325.997} C_VEL
LIN {X 0,Y 432.349,Z 733.44,A -85,B 0,C 180,E1 -9329.49,E2 -9329.49} C_VEL
LIN {X 0,Y 432.392,Z 733.43,A -85,B 0,C 180,E1 -9332.928,E2 -9332.928} C_VEL
LIN {X 0,Y 432.372,Z 733.431,A -85,B 0,C 180,E1 -9336.023,E2 -9336.023} C_VEL
LIN {X 0,Y 432.352,Z 733.445,A -85,B 0,C 180,E1 -9339.046,E2 -9339.046} C_VEL
LIN {X 0,Y 432.363,Z 733.425,A -85,B 0,C 180,E1 -9342.01,E2 -9342.01} C_VEL
LIN {X 0,Y 432.398,Z 733.428,A -85,B 0,C 180,E1 -9344.926,E2 -9344.926} C_VEL
LIN {X 0,Y 432.461,Z 733.426,A -85,B 0,C 180,E1 -9347.803,E2 -9347.803} C_VEL
LIN {X 0,Y 432.494,Z 733.408,A -85,B 0,C 180,E1 -9351.59,E2 -9351.59} C_VEL
LIN {X 0,Y 432.597,Z 733.4,A -85,B 0,C 180,E1 -9354.406,E2 -9354.406} C_VEL
LIN {X 0,Y 432.608,Z 733.405,A -85,B 0,C 180,E1 -9358.138,E2 -9358.138} C_VEL
LIN {X 0,Y 432.734,Z 733.385,A -85,B 0,C 180,E1 -9360,E2 -9360} C_VEL
LIN {X 0,Y 432.594,Z 733.391,A -85,B 0,C 180,E1 -9362.794,E2 -9362.794} C_VEL
LIN {X 0,Y 432.568,Z 733.411,A -85,B 0,C 180,E1 -9366.53,E2 -9366.53} C_VEL
LIN {X 0,Y 432.445,Z 733.428,A -85,B 0,C 180,E1 -9369.353,E2 -9369.353} C_VEL
LIN {X 0,Y 432.432,Z 733.414,A -85,B 0,C 180,E1 -9372.803,E2 -9372.803} C_VEL
LIN {X 0,Y 432.414,Z 733.431,A -85,B 0,C 180,E1 -9376.479,E2 -9376.479} C_VEL
LIN {X 0,Y 432.375,Z 733.43,A -85,B 0,C 180,E1 -9379.959,E2 -9379.959} C_VEL
LIN {X 0,Y 432.321,Z 733.436,A -85,B 0,C 180,E1 -9382.964,E2 -9382.964} C_VEL
LIN {X 0,Y 432.366,Z 733.443,A -85,B 0,C 180,E1 -9386.032,E2 -9386.032} C_VEL
LIN {X 0,Y 432.344,Z 733.429,A -85,B 0,C 180,E1 -9389.187,E2 -9389.187} C_VEL
LIN {X 0,Y 432.324,Z 733.446,A -85,B 0,C 180,E1 -9392.443,E2 -9392.443} C_VEL
LIN {X 0,Y 432.347,Z 733.436,A -85,B 0,C 180,E1 -9395.632,E2 -9395.632} C_VEL
LIN {X 0,Y 432.359,Z 733.405,A -85,B 0,C 180,E1 -9398.717,E2 -9398.717} C_VEL
LIN {X 0,Y 432.366,Z 733.424,A -85,B 0,C 180,E1 -9401.793,E2 -9401.793} C_VEL
LIN {X 0,Y 432.334,Z 733.445,A -85,B 0,C 180,E1 -9404.347,E2 -9404.347} C_VEL
LIN {X 0,Y 432.323,Z 733.436,A -85,B 0,C 180,E1 -9407.015,E2 -9407.015} C_VEL
LIN {X 0,Y 432.344,Z 733.433,A -85,B 0,C 180,E1 -9409.819,E2 -9409.819} C_VEL
LIN {X 0,Y 432.317,Z 733.44,A -85,B 0,C 180,E1 -9413.023,E2 -9413.023} C_VEL
LIN {X 0,Y 432.36,Z 733.439,A -85,B 0,C 180,E1 -9415.996,E2 -9415.996} C_VEL
LIN {X 0,Y 432.348,Z 733.424,A -85,B 0,C 180,E1 -9419.489,E2 -9419.489} C_VEL
LIN {X 0,Y 432.393,Z 733.429,A -85,B 0,C 180,E1 -9422.928,E2 -9422.928} C_VEL
LIN {X 0,Y 432.417,Z 733.5,A -85,B 0,C 180,E1 -9425.425,E2 -9425.425} C_VEL
LIN {X 0,Y 434.042,Z 743.064,A -85,B 0,C 180,E1 -9427.782,E2 -9427.782} C_VEL
LIN {X 0,Y 433.502,Z 754.365,A -85,B 0,C 180,E1 -9430.342,E2 -9430.342} C_VEL
LIN {X 0,Y 432.841,Z 767.677,A -85,B 0,C 180,E1 -9433.331,E2 -9433.331} C_VEL
LIN {X 0,Y 432.446,Z 777.581,A -85,B 0,C 180,E1 -9435.485,E2 -9435.485} C_VEL
LIN {X 0,Y 433.351,Z 784.635,A -85,B 0,C 180,E1 -9435.673,E2 -9435.673} C_VEL
LIN {X 0,Y 434.982,Z 797.881,A -85,B 0,C 180,E1 -9435.948,E2 -9435.948} C_VEL
LIN {X 0,Y 434.663,Z 853.529,A -85,B 0,C 180,E1 -9436.884,E2 -9436.884} C_VEL
LIN {X 0,Y 434.371,Z 862.932,A -85,B 0,C 180,E1 -9437.146,E2 -9437.146} C_VEL
LIN {X 0,Y 434.053,Z 871.405,A -85,B 0,C 180,E1 -9437.493,E2 -9437.493} C_VEL
LIN {X 0,Y 433.721,Z 879.919,A -85,B 0,C 180,E1 -9437.958,E2 -9437.958} C_VEL
LIN {X 0,Y 433.361,Z 888.266,A -85,B 0,C 180,E1 -9438.541,E2 -9438.541} C_VEL
LIN {X 0,Y 432.974,Z 896.321,A -85,B 0,C 180,E1 -9439.242,E2 -9439.242} C_VEL
LIN {X 0,Y 432.475,Z 905.015,A -85,B 0,C 180,E1 -9440.175,E2 -9440.175} C_VEL
LIN {X 0,Y 432.034,Z 913.549,A -85,B 0,C 180,E1 -9441.346,E2 -9441.346} C_VEL
LIN {X 0,Y 431.734,Z 920.248,A -85,B 0,C 180,E1 -9442.517,E2 -9442.517} C_VEL
LIN {X 0,Y 431.521,Z 924.647,A -85,B 0,C 180,E1 -9443.454,E2 -9443.454} C_VEL
LIN {X 0,Y 431.398,Z 928.308,A -85,B 0,C 180,E1 -9444.391,E2 -9444.391} C_VEL
LIN {X 0,Y 431.32,Z 931.313,A -85,B 0,C 180,E1 -9445.327,E2 -9445.327} C_VEL
LIN {X 0,Y 431.237,Z 933.643,A -85,B 0,C 180,E1 -9446.262,E2 -9446.262} C_VEL
LIN {X 0,Y 431.24,Z 935.396,A -85,B 0,C 180,E1 -9447.198,E2 -9447.198} C_VEL
LIN {X 0,Y 431.199,Z 936.651,A -85,B 0,C 180,E1 -9448.132,E2 -9448.132} C_VEL
LIN {X 0,Y 431.166,Z 937.433,A -85,B 0,C 180,E1 -9449.066,E2 -9449.066} C_VEL
LIN {X 0,Y 431.164,Z 937.729,A -85,B 0,C 180,E1 -9450,E2 -9450} C_VEL
LIN {X 0,Y 431.166,Z 937.432,A -85,B 0,C 180,E1 -9450.934,E2 -9450.934} C_VEL
LIN {X 0,Y 431.199,Z 936.649,A -85,B 0,C 180,E1 -9451.868,E2 -9451.868} C_VEL
LIN {X 0,Y 431.24,Z 935.393,A -85,B 0,C 180,E1 -9452.802,E2 -9452.802} C_VEL
LIN {X 0,Y 431.263,Z 932.481,A -85,B 0,C 180,E1 -9454.205,E2 -9454.205} C_VEL
LIN {X 0,Y 431.376,Z 929.829,A -85,B 0,C 180,E1 -9455.141,E2 -9455.141} C_VEL
LIN {X 0,Y 431.45,Z 926.102,A -85,B 0,C 180,E1 -9456.189,E2 -9456.189} C_VEL
LIN {X 0,Y 431.653,Z 921.412,A -85,B 0,C 180,E1 -9457.249,E2 -9457.249} C_VEL
LIN {X 0,Y 431.894,Z 916.384,A -85,B 0,C 180,E1 -9458.186,E2 -9458.186} C_VEL
LIN {X 0,Y 432.194,Z 910.327,A -85,B 0,C 180,E1 -9459.123,E2 -9459.123} C_VEL
LIN {X 0,Y 432.599,Z 902.96,A -85,B 0,C 180,E1 -9460.058,E2 -9460.058} C_VEL
LIN {X 0,Y 433.014,Z 895.072,A -85,B 0,C 180,E1 -9460.876,E2 -9460.876} C_VEL
LIN {X 0,Y 433.421,Z 886.738,A -85,B 0,C 180,E1 -9461.576,E2 -9461.576} C_VEL
LIN {X 0,Y 433.981,Z 876.105,A -85,B 0,C 180,E1 -9462.272,E2 -9462.272} C_VEL
LIN {X 0,Y 434.249,Z 864.539,A -85,B 0,C 180,E1 -9462.798,E2 -9462.798} C_VEL
LIN {X 0,Y 434.596,Z 854.879,A -85,B 0,C 180,E1 -9463.085,E2 -9463.085} C_VEL
LIN {X 0,Y 434.865,Z 795.691,A -85,B 0,C 180,E1 -9464.09,E2 -9464.09} C_VEL
LIN {X 0,Y 432.466,Z 777.971,A -85,B 0,C 180,E1 -9464.482,E2 -9464.482} C_VEL
LIN {X 0,Y 432.488,Z 776.034,A -85,B 0,C 180,E1 -9464.805,E2 -9464.805} C_VEL
LIN {X 0,Y 433.182,Z 760.848,A -85,B 0,C 180,E1 -9468.199,E2 -9468.199} C_VEL
LIN {X 0,Y 433.995,Z 745.68,A -85,B 0,C 180,E1 -9471.617,E2 -9471.617} C_VEL
LIN {X 0,Y 433.864,Z 741.515,A -85,B 0,C 180,E1 -9472.584,E2 -9472.584} C_VEL
LIN {X 0,Y 432.417,Z 733.499,A -85,B 0,C 180,E1 -9474.575,E2 -9474.575} C_VEL
LIN {X 0,Y 432.393,Z 733.429,A -85,B 0,C 180,E1 -9477.072,E2 -9477.072} C_VEL
LIN {X 0,Y 432.348,Z 733.425,A -85,B 0,C 180,E1 -9480.511,E2 -9480.511} C_VEL
LIN {X 0,Y 432.36,Z 733.44,A -85,B 0,C 180,E1 -9484.004,E2 -9484.004} C_VEL
LIN {X 0,Y 432.333,Z 733.441,A -85,B 0,C 180,E1 -9487.199,E2 -9487.199} C_VEL
LIN {X 0,Y 432.344,Z 733.432,A -85,B 0,C 180,E1 -9490.181,E2 -9490.181} C_VEL
LIN {X 0,Y 432.321,Z 733.437,A -85,B 0,C 180,E1 -9493.061,E2 -9493.061} C_VEL
LIN {X 0,Y 432.333,Z 733.445,A -85,B 0,C 180,E1 -9495.665,E2 -9495.665} C_VEL
LIN {X 0,Y 432.367,Z 733.422,A -85,B 0,C 180,E1 -9498.393,E2 -9498.393} C_VEL
LIN {X 0,Y 432.352,Z 733.414,A -85,B 0,C 180,E1 -9501.852,E2 -9501.852} C_VEL
LIN {X 0,Y 432.342,Z 733.438,A -85,B 0,C 180,E1 -9505.323,E2 -9505.323} C_VEL
LIN {X 0,Y 432.322,Z 733.438,A -85,B 0,C 180,E1 -9508.654,E2 -9508.654} C_VEL
LIN {X 0,Y 432.384,Z 733.432,A -85,B 0,C 180,E1 -9511.877,E2 -9511.877} C_VEL
LIN {X 0,Y 432.353,Z 733.437,A -85,B 0,C 180,E1 -9514.999,E2 -9514.999} C_VEL
LIN {X 0,Y 432.36,Z 733.43,A -85,B 0,C 180,E1 -9518.046,E2 -9518.046} C_VEL
LIN {X 0,Y 432.388,Z 733.43,A -85,B 0,C 180,E1 -9521.03,E2 -9521.03} C_VEL
LIN {X 0,Y 432.432,Z 733.433,A -85,B 0,C 180,E1 -9523.961,E2 -9523.961} C_VEL
LIN {X 0,Y 432.461,Z 733.413,A -85,B 0,C 180,E1 -9527.804,E2 -9527.804} C_VEL
LIN {X 0,Y 432.494,Z 733.419,A -85,B 0,C 180,E1 -9531.59,E2 -9531.59} C_VEL
LIN {X 0,Y 432.597,Z 733.41,A -85,B 0,C 180,E1 -9534.406,E2 -9534.406} C_VEL
LIN {X 0,Y 432.606,Z 733.392,A -85,B 0,C 180,E1 -9538.138,E2 -9538.138} C_VEL
LIN {X 0,Y 432.736,Z 733.384,A -85,B 0,C 180,E1 -9540,E2 -9540} C_VEL
LIN {X 0,Y 432.608,Z 733.41,A -85,B 0,C 180,E1 -9542.794,E2 -9542.794} C_VEL
LIN {X 0,Y 432.571,Z 733.403,A -85,B 0,C 180,E1 -9546.53,E2 -9546.53} C_VEL
LIN {X 0,Y 432.444,Z 733.421,A -85,B 0,C 180,E1 -9549.353,E2 -9549.353} C_VEL
LIN {X 0,Y 432.433,Z 733.435,A -85,B 0,C 180,E1 -9552.804,E2 -9552.804} C_VEL
LIN {X 0,Y 432.414,Z 733.425,A -85,B 0,C 180,E1 -9556.479,E2 -9556.479} C_VEL
LIN {X 0,Y 432.34,Z 733.437,A -85,B 0,C 180,E1 -9559.96,E2 -9559.96} C_VEL
LIN {X 0,Y 432.32,Z 733.446,A -85,B 0,C 180,E1 -9562.964,E2 -9562.964} C_VEL
LIN {X 0,Y 432.363,Z 733.424,A -85,B 0,C 180,E1 -9566.033,E2 -9566.033} C_VEL
LIN {X 0,Y 432.344,Z 733.446,A -85,B 0,C 180,E1 -9569.187,E2 -9569.187} C_VEL
LIN {X 0,Y 432.323,Z 733.437,A -85,B 0,C 180,E1 -9572.443,E2 -9572.443} C_VEL
LIN {X 0,Y 432.344,Z 733.442,A -85,B 0,C 180,E1 -9575.632,E2 -9575.632} C_VEL
LIN {X 0,Y 432.342,Z 733.439,A -85,B 0,C 180,E1 -9578.714,E2 -9578.714} C_VEL
LIN {X 0,Y 432.326,Z 733.412,A -85,B 0,C 180,E1 -9581.798,E2 -9581.798} C_VEL
LIN {X 0,Y 432.335,Z 733.428,A -85,B 0,C 180,E1 -9584.347,E2 -9584.347} C_VEL
LIN {X 0,Y 432.321,Z 733.443,A -85,B 0,C 180,E1 -9587.016,E2 -9587.016} C_VEL
LIN {X 0,Y 432.334,Z 733.435,A -85,B 0,C 180,E1 -9589.821,E2 -9589.821} C_VEL
LIN {X 0,Y 432.307,Z 733.437,A -85,B 0,C 180,E1 -9593.022,E2 -9593.022} C_VEL
LIN {X 0,Y 432.359,Z 733.441,A -85,B 0,C 180,E1 -9595.997,E2 -9595.997} C_VEL
LIN {X 0,Y 432.347,Z 733.436,A -85,B 0,C 180,E1 -9599.49,E2 -9599.49} C_VEL
LIN {X 0,Y 432.348,Z 733.442,A -85,B 0,C 180,E1 -9601.874,E2 -9601.874} C_VEL
LIN {X 0,Y 432.379,Z 733.44,A -85,B 0,C 180,E1 -9605.539,E2 -9605.539} C_VEL
LIN {X 0,Y 432.361,Z 733.439,A -85,B 0,C 180,E1 -9609.047,E2 -9609.047} C_VEL
LIN {X 0,Y 432.424,Z 733.536,A -85,B 0,C 180,E1 -9609.92,E2 -9609.92} C_VEL
LIN {X 0,Y 432.997,Z 737.365,A -85,B 0,C 180,E1 -9611.057,E2 -9611.057} C_VEL
LIN {X 0,Y 432.829,Z 745.564,A -85,B 0,C 180,E1 -9613.337,E2 -9613.337} C_VEL
LIN {X 0,Y 432.478,Z 753.933,A -85,B 0,C 180,E1 -9615.54,E2 -9615.54} C_VEL
LIN {X 0,Y 433.247,Z 758.35,A -85,B 0,C 180,E1 -9615.69,E2 -9615.69} C_VEL
LIN {X 0,Y 435.127,Z 768.92,A -85,B 0,C 180,E1 -9615.931,E2 -9615.931} C_VEL
LIN {X 0,Y 434.677,Z 829.296,A -85,B 0,C 180,E1 -9616.947,E2 -9616.947} C_VEL
LIN {X 0,Y 434.525,Z 839.181,A -85,B 0,C 180,E1 -9617.239,E2 -9617.239} C_VEL
LIN {X 0,Y 434.117,Z 850.325,A -85,B 0,C 180,E1 -9617.732,E2 -9617.732} C_VEL
LIN {X 0,Y 433.737,Z 861.404,A -85,B 0,C 180,E1 -9618.451,E2 -9618.451} C_VEL
LIN {X 0,Y 432.862,Z 866.617,A -85,B 0,C 180,E1 -9618.841,E2 -9618.841} C_VEL
LIN {X 0,Y 429.592,Z 874.612,A -85,B 0,C 180,E1 -9619.523,E2 -9619.523} C_VEL
LIN {X 0,Y 426.342,Z 881.866,A -85,B 0,C 180,E1 -9620.298,E2 -9620.298} C_VEL
LIN {X 0,Y 425.435,Z 885.864,A -85,B 0,C 180,E1 -9620.84,E2 -9620.84} C_VEL
LIN {X 0,Y 424.987,Z 893.858,A -85,B 0,C 180,E1 -9622.159,E2 -9622.159} C_VEL
LIN {X 0,Y 424.809,Z 899.427,A -85,B 0,C 180,E1 -9623.35,E2 -9623.35} C_VEL
LIN {X 0,Y 424.418,Z 904.608,A -85,B 0,C 180,E1 -9624.775,E2 -9624.775} C_VEL
LIN {X 0,Y 424.345,Z 907.266,A -85,B 0,C 180,E1 -9625.726,E2 -9625.726} C_VEL
LIN {X 0,Y 424.269,Z 910.175,A -85,B 0,C 180,E1 -9627.152,E2 -9627.152} C_VEL
LIN {X 0,Y 424.152,Z 911.45,A -85,B 0,C 180,E1 -9628.101,E2 -9628.101} C_VEL
LIN {X 0,Y 424.089,Z 912.256,A -85,B 0,C 180,E1 -9629.05,E2 -9629.05} C_VEL
LIN {X 0,Y 424.083,Z 912.562,A -85,B 0,C 180,E1 -9630,E2 -9630} C_VEL
LIN {X 0,Y 424.09,Z 912.287,A -85,B 0,C 180,E1 -9630.95,E2 -9630.95} C_VEL
LIN {X 0,Y 424.152,Z 911.544,A -85,B 0,C 180,E1 -9631.899,E2 -9631.899} C_VEL
LIN {X 0,Y 424.269,Z 910.332,A -85,B 0,C 180,E1 -9632.848,E2 -9632.848} C_VEL
LIN {X 0,Y 424.34,Z 907.489,A -85,B 0,C 180,E1 -9634.274,E2 -9634.274} C_VEL
LIN {X 0,Y 424.413,Z 904.901,A -85,B 0,C 180,E1 -9635.226,E2 -9635.226} C_VEL
LIN {X 0,Y 424.752,Z 899.8,A -85,B 0,C 180,E1 -9636.651,E2 -9636.651} C_VEL
LIN {X 0,Y 425.005,Z 893.105,A -85,B 0,C 180,E1 -9638.08,E2 -9638.08} C_VEL
LIN {X 0,Y 425.475,Z 885.748,A -85,B 0,C 180,E1 -9639.268,E2 -9639.268} C_VEL
LIN {X 0,Y 425.919,Z 878.487,A -85,B 0,C 180,E1 -9640.217,E2 -9640.217} C_VEL
LIN {X 0,Y 426.336,Z 870.727,A -85,B 0,C 180,E1 -9641.048,E2 -9641.048} C_VEL
LIN {X 0,Y 426.634,Z 864.038,A -85,B 0,C 180,E1 -9641.642,E2 -9641.642} C_VEL
LIN {X 0,Y 427.008,Z 855.862,A -85,B 0,C 180,E1 -9642.234,E2 -9642.234} C_VEL
LIN {X 0,Y 427.394,Z 847.577,A -85,B 0,C 180,E1 -9642.705,E2 -9642.705} C_VEL
LIN {X 0,Y 427.649,Z 838.631,A -85,B 0,C 180,E1 -9643.09,E2 -9643.09} C_VEL
LIN {X 0,Y 427.803,Z 829.31,A -85,B 0,C 180,E1 -9643.364,E2 -9643.364} C_VEL
LIN {X 0,Y 428.208,Z 769.655,A -85,B 0,C 180,E1 -9644.386,E2 -9644.386} C_VEL
LIN {X 0,Y 425.476,Z 753.977,A -85,B 0,C 180,E1 -9644.773,E2 -9644.773} C_VEL
LIN {X 0,Y 425.966,Z 743.12,A -85,B 0,C 180,E1 -9647.772,E2 -9647.772} C_VEL
LIN {X 0,Y 425.939,Z 737.859,A -85,B 0,C 180,E1 -9649.269,E2 -9649.269} C_VEL
LIN {X 0,Y 425.387,Z 734.389,A -85,B 0,C 180,E1 -9650.364,E2 -9650.364} C_VEL
LIN {X 0,Y 425.346,Z 734.316,A -85,B 0,C 180,E1 -9654.398,E2 -9654.398} C_VEL
LIN {X 0,Y 425.271,Z 734.322,A -85,B 0,C 180,E1 -9657.563,E2 -9657.563} C_VEL
LIN {X 0,Y 425.291,Z 734.314,A -85,B 0,C 180,E1 -9660.761,E2 -9660.761} C_VEL
LIN {X 0,Y 425.311,Z 734.321,A -85,B 0,C 180,E1 -9664.288,E2 -9664.288} C_VEL
LIN {X 0,Y 425.278,Z 734.312,A -85,B 0,C 180,E1 -9667.694,E2 -9667.694} C_VEL
LIN {X 0,Y 425.281,Z 734.317,A -85,B 0,C 180,E1 -9670.52,E2 -9670.52} C_VEL
LIN {X 0,Y 425.258,Z 734.321,A -85,B 0,C 180,E1 -9673.351,E2 -9673.351} C_VEL
LIN {X 0,Y 425.256,Z 734.298,A -85,B 0,C 180,E1 -9676.649,E2 -9676.649} C_VEL
LIN {X 0,Y 425.286,Z 734.306,A -85,B 0,C 180,E1 -9679.872,E2 -9679.872} C_VEL
LIN {X 0,Y 425.279,Z 734.321,A -85,B 0,C 180,E1 -9682.488,E2 -9682.488} C_VEL
LIN {X 0,Y 425.307,Z 734.309,A -85,B 0,C 180,E1 -9685.817,E2 -9685.817} C_VEL
LIN {X 0,Y 425.292,Z 734.321,A -85,B 0,C 180,E1 -9689.239,E2 -9689.239} C_VEL
LIN {X 0,Y 425.35,Z 734.309,A -85,B 0,C 180,E1 -9692.442,E2 -9692.442} C_VEL
LIN {X 0,Y 425.351,Z 734.307,A -85,B 0,C 180,E1 -9695.602,E2 -9695.602} C_VEL
LIN {X 0,Y 425.295,Z 734.32,A -85,B 0,C 180,E1 -9698.681,E2 -9698.681} C_VEL
LIN {X 0,Y 425.324,Z 734.303,A -85,B 0,C 180,E1 -9701.702,E2 -9701.702} C_VEL
LIN {X 0,Y 425.351,Z 734.303,A -85,B 0,C 180,E1 -9704.671,E2 -9704.671} C_VEL
LIN {X 0,Y 425.414,Z 734.305,A -85,B 0,C 180,E1 -9707.598,E2 -9707.598} C_VEL
LIN {X 0,Y 425.444,Z 734.287,A -85,B 0,C 180,E1 -9711.45,E2 -9711.45} C_VEL
LIN {X 0,Y 425.553,Z 734.278,A -85,B 0,C 180,E1 -9714.313,E2 -9714.313} C_VEL
LIN {X 0,Y 425.578,Z 734.281,A -85,B 0,C 180,E1 -9718.107,E2 -9718.107} C_VEL
LIN {X 0,Y 425.703,Z 734.26,A -85,B 0,C 180,E1 -9720,E2 -9720} C_VEL
LIN {X 0,Y 425.548,Z 734.268,A -85,B 0,C 180,E1 -9722.84,E2 -9722.84} C_VEL
LIN {X 0,Y 425.526,Z 734.288,A -85,B 0,C 180,E1 -9726.639,E2 -9726.639} C_VEL
LIN {X 0,Y 425.403,Z 734.307,A -85,B 0,C 180,E1 -9729.509,E2 -9729.509} C_VEL
LIN {X 0,Y 425.395,Z 734.291,A -85,B 0,C 180,E1 -9732.904,E2 -9732.904} C_VEL
LIN {X 0,Y 425.363,Z 734.309,A -85,B 0,C 180,E1 -9736.605,E2 -9736.605} C_VEL
LIN {X 0,Y 425.362,Z 734.309,A -85,B 0,C 180,E1 -9739.648,E2 -9739.648} C_VEL
LIN {X 0,Y 425.309,Z 734.311,A -85,B 0,C 180,E1 -9743.365,E2 -9743.365} C_VEL
LIN {X 0,Y 425.349,Z 734.309,A -85,B 0,C 180,E1 -9746.844,E2 -9746.844} C_VEL
LIN {X 0,Y 425.292,Z 734.309,A -85,B 0,C 180,E1 -9749.719,E2 -9749.719} C_VEL
LIN {X 0,Y 425.283,Z 734.319,A -85,B 0,C 180,E1 -9753.048,E2 -9753.048} C_VEL
LIN {X 0,Y 425.286,Z 734.316,A -85,B 0,C 180,E1 -9755.929,E2 -9755.929} C_VEL
LIN {X 0,Y 425.311,Z 734.28,A -85,B 0,C 180,E1 -9759.045,E2 -9759.045} C_VEL
LIN {X 0,Y 425.316,Z 734.303,A -85,B 0,C 180,E1 -9761.962,E2 -9761.962} C_VEL
LIN {X 0,Y 425.287,Z 734.318,A -85,B 0,C 180,E1 -9765.283,E2 -9765.283} C_VEL
LIN {X 0,Y 425.276,Z 734.31,A -85,B 0,C 180,E1 -9768.621,E2 -9768.621} C_VEL
LIN {X 0,Y 425.318,Z 734.317,A -85,B 0,C 180,E1 -9771.103,E2 -9771.103} C_VEL
LIN {X 0,Y 425.301,Z 734.315,A -85,B 0,C 180,E1 -9774.664,E2 -9774.664} C_VEL
LIN {X 0,Y 425.266,Z 734.317,A -85,B 0,C 180,E1 -9778.073,E2 -9778.073} C_VEL
LIN {X 0,Y 425.332,Z 734.317,A -85,B 0,C 180,E1 -9781.368,E2 -9781.368} C_VEL
LIN {X 0,Y 425.32,Z 734.318,A -85,B 0,C 180,E1 -9784.556,E2 -9784.556} C_VEL
LIN {X 0,Y 425.396,Z 734.556,A -85,B 0,C 180,E1 -9785.32,E2 -9785.32} C_VEL
LIN {X 0,Y 427.072,Z 744.424,A -85,B 0,C 180,E1 -9787.76,E2 -9787.76} C_VEL
LIN {X 0,Y 426.47,Z 755.565,A -85,B 0,C 180,E1 -9790.324,E2 -9790.324} C_VEL
LIN {X 0,Y 425.783,Z 768.764,A -85,B 0,C 180,E1 -9793.339,E2 -9793.339} C_VEL
LIN {X 0,Y 425.408,Z 777.244,A -85,B 0,C 180,E1 -9795.225,E2 -9795.225} C_VEL
LIN {X 0,Y 425.833,Z 780.607,A -85,B 0,C 180,E1 -9795.349,E2 -9795.349} C_VEL
LIN {X 0,Y 428.082,Z 797.689,A -85,B 0,C 180,E1 -9795.716,E2 -9795.716} C_VEL
LIN {X 0,Y 427.682,Z 854.772,A -85,B 0,C 180,E1 -9796.699,E2 -9796.699} C_VEL
LIN {X 0,Y 427.379,Z 865.227,A -85,B 0,C 180,E1 -9797.022,E2 -9797.022} C_VEL
LIN {X 0,Y 426.988,Z 875.93,A -85,B 0,C 180,E1 -9797.524,E2 -9797.524} C_VEL
LIN {X 0,Y 426.466,Z 886.557,A -85,B 0,C 180,E1 -9798.233,E2 -9798.233} C_VEL
LIN {X 0,Y 426.039,Z 894.882,A -85,B 0,C 180,E1 -9798.944,E2 -9798.944} C_VEL
LIN {X 0,Y 425.597,Z 902.762,A -85,B 0,C 180,E1 -9799.775,E2 -9799.775} C_VEL
LIN {X 0,Y 425.191,Z 910.131,A -85,B 0,C 180,E1 -9800.726,E2 -9800.726} C_VEL
LIN {X 0,Y 424.788,Z 917.609,A -85,B 0,C 180,E1 -9801.916,E2 -9801.916} C_VEL
LIN {X 0,Y 424.459,Z 924.439,A -85,B 0,C 180,E1 -9803.344,E2 -9803.344} C_VEL
LIN {X 0,Y 424.292,Z 929.626,A -85,B 0,C 180,E1 -9804.773,E2 -9804.773} C_VEL
LIN {X 0,Y 424.185,Z 932.277,A -85,B 0,C 180,E1 -9805.724,E2 -9805.724} C_VEL
